# B&R Automation Studio project NAEUL004C00R13L518F00 (part 49)

#### Act_Main.st
```iecst
(** 2019-01-20 **)
ACTION Act_Main:

	IF eStatOld <> eStat THEN

		fbTxInTimer(IN := FALSE);
		fbTxOutTimer(IN := FALSE);
		fbMagOutTrig(CLK := FALSE);

		bMcRunRdy				 	  := FALSE;
		bRdyEnt			 		   	  := FALSE;
		bRdyExit				  	  := FALSE;
		bMagConvRun    := FALSE;
		fbCheckErrorTim(IN:= FALSE);
		usiStep		:= 0;

		sStatTxt	:= a_sStatText[eStat];

		eStatOld	:= eStat;

		eStatus		:= Busy;
	END_IF

	//Main
	CASE eStat OF

		AGVMagActIdle:
			eStatus	:= Idle;
			bMagConvRdy := FALSE;

		AGVMagActEnter:

			IF eStatus = Idle OR eStatus = Busy THEN

				eStatus	:= Busy;
				bMagConvRdy := TRUE;

				IF usiStep = 0 THEN

					IF bAIVAuto AND bMagConvAuto
						OR p_bSOTAvailable
						THEN // ON Connection

						bMagConvRdy  := TRUE; //Allow VEH to Move In

						IF bAIVInPos OR p_bSOTRcvOk THEN // VEH is in Position to Enter

							bRdyEnt := TRUE;

						END_IF
					END_IF

						IF bRdyEnt THEN

							IF bAIVInPos OR p_bSOTRcvOk  THEN

								bMagConvRdy := FALSE; // Temporarily Not Allowed Other VEH while one VEH in Pos.

								IF p_bSOTErr THEN
									eStatus		:= Error;
									udiStatus	:= 10010;//SOT Sensor Error Has Been Activated;

								ELSIF (NOT bMagConvOccupied) (*AND p_tyAGVToDTMag.bVEHOccupied*) THEN

									bMcRunRdy	:= TRUE;

									bMagConvRun := TRUE;

									usiStep	:= 1;
								ELSE
									eStatus		:= Error;
									udiStatus	:= 10000;	//Magazine Is Present Before Entering
								END_IF

							ELSE
								eStatus		:= Error;
								udiStatus	:= 10001;	//AIV Not In Enter Position
							END_IF

						END_IF

				ELSIF usiStep = 1 THEN

					IF p_eDirection = ConvDirLToL OR p_eDirection = ConvDirLToR THEN
						bEndSen	:= p_bMagConvRgtSen;
					ELSE
						bEndSen	:= p_bMagConvLftSen;
					END_IF

					fbTxInTimer(IN := TRUE, PT := DINT_TO_TIME(p_diTxInTimeOut));

					IF bEndSen = TRUE (*AND p_tyAGVToDTMag.bVEHOccupied = FALSE*) THEN

						eStatus	:= Done;

						bMagConvRdy := TRUE; // Allow VEH to Move Out After Transfering Magazine

						bMagConvRun := FALSE;

					ELSIF fbTxInTimer.Q = TRUE THEN

						eStatus		:= Error;
						udiStatus	:= 10002;	//Transfer In Time Out While Transporting

					END_IF

					IF bAIVInPos = FALSE AND p_bSOTRcvOk = FALSE AND eStatus = Busy THEN

						eStatus		:= Error;
						udiStatus	:= 10001;	//AIV Not In Enter Position
					END_IF

//					IF bAIVAuto = FALSE AND eStatus = Busy THEN
//
//						eStatus		:= Error;
//						udiStatus	:= 10006;	//AIV Not In Enter Position
//					END_IF
				END_IF

			END_IF

		AGVMagActExit:
			IF eStatus = Idle OR eStatus = Busy THEN

				eStatus	:= Busy;

				bMagConvRdy := TRUE;

				IF usiStep = 0 THEN

					IF bAIVAuto AND bMagConvAuto
						OR p_bSOTRdy
						THEN // ON Connection

						bMagConvRdy  := TRUE; //Allow VEH to Move In

						IF bAIVInPos OR p_bSOTRcvOk THEN // VEH is in Position to Exit

							bRdyExit := TRUE;

						END_IF
					END_IF

						IF bRdyExit THEN

							IF (bAIVInPos OR p_bSOTRcvOk) AND bAIVOccupied=FALSE THEN

								bMagConvRdy := FALSE; // Temporarily Not Allowed Other VEH while one VEH in Pos.

								IF bMagConvOccupied OR p_bSOTRdy = FALSE THEN

									bMcRunRdy	:= TRUE;

									bMagConvRun := TRUE;

									usiStep	:= 1;

								ELSE
									eStatus		:= Error;
									udiStatus	:= 10003;	//Magazine Is Not Present Before Exiting
								END_IF

							ELSE
								eStatus		:= Error;
								udiStatus	:= 10004;	//AIV Not In Exit Position
							END_IF
						END_IF

				ELSIF usiStep = 1 THEN

					IF p_bSOTErr THEN

						usiStep := 2;
					END_IF

					IF p_eDirection = ConvDirLToR OR p_eDirection = ConvDirRToR THEN
						bEndSen	:= p_bMagConvRgtSen;
					ELSE
						bEndSen	:= p_bMagConvLftSen;
					END_IF

					fbTxOutTimer(IN := TRUE, PT := DINT_TO_TIME(p_diTxOutTimeOut));

					IF bEndSen = FALSE AND (bAIVOccupied = TRUE OR p_bSOTRdy = FALSE) THEN

						usiStep := 2;

					ELSIF fbTxOutTimer.Q = TRUE THEN

						eStatus		:= Error;
						udiStatus	:= 10005;	//Transfer Out Time Out While Transporting

					END_IF

					IF bAIVInPos = FALSE AND p_bSOTRcvOk = FALSE AND eStatus = Busy THEN

						eStatus		:= Error;
						udiStatus	:= 10001;	//AIV Not In Enter Position
					END_IF

//					IF bAIVAuto = FALSE AND eStatus = Busy THEN
//
//						eStatus		:= Error;
//						udiStatus	:= 10006;	//AIV Not In Auto
//					END_IF

				ELSIF usiStep = 2 THEN
					fbCheckErrorTim(IN:= TRUE);
					IF p_bSOTErr THEN
						eStatus		:= Error;
						udiStatus	:= 10010;	//SOT Error signal activated
					ELSIF fbCheckErrorTim.Q THEN
						usiStep := 3;
					END_IF

				ELSIF usiStep = 3 THEN
					bMagConvRdy 	   := TRUE; // Allow VEH to Move Out After Transfering Magazine

					bMagConvRun := FALSE;
					eStatus := Done;
				END_IF

			END_IF
	END_CASE

END_ACTION
```

#### Act_OutputConfig.st
```iecst
ACTION Act_OutputConfig:

	g_tyAGV2 := tylocalAGV.Out; // Change the Global Naming According to the Physical Hardware Module

END_ACTION
```

#### Cyclic.st
```iecst
(** 2019-01-11 **)
PROGRAM _CYCLIC

	IF bInitialDone = FALSE THEN
		IF g_tyStartUp.bNtSettingsLoadDone = TRUE THEN
			bInitialDone	:= TRUE;
			Act_Initial;
		END_IF

	ELSE
		Act_InputConfig;
		IF (tylocalAGV.In.bPrep = TRUE) AND (tylocalAGV.In.bEn = TRUE) AND (tylocalAGV.In.bDis = FALSE) THEN
			Act_Link;
			Act_Background;
			Act_Main;
		ELSE
			IF tylocalAGV.Out.eStat <> AGVMagActIdle THEN
				eStatus	:= Done;
			ELSE
				eStatus	:= Idle;
			END_IF
		END_IF
		Act_OutputConfig;
		Act_Alarm;

	END_IF

END_PROGRAM
```

#### Init.st
```iecst
(** 2019-01-20 **)
PROGRAM _INIT

	(* Always Change If Project Change *)

	sProgNm	:= 'AGVMag 2';

	//Physical Configuration

	//Pass Address To Global Address For External Use
	//Action, State & Status
	p_AGVMag2Stat				:= ADR(eStat);
	p_AGVMag2Status				:= ADR(eStatus);
	p_AGVMag2StatTxt			:= ADR(sStatTxt);

	//Alarm
	p_AGVMag2AlmData			:= ADR(tyAlmData);

	//Output
	p_AGVMag2RdyEnter			:= ADR(bRdyEnt);
	p_AGVMag2RdyExit			:= ADR(bRdyExit);
	p_AGVMag2McRunRdy			:= ADR(bMcRunRdy);
	p_AGVMag2DTMagToAGV			:= ADR(tyDTMagToAGV);

	(* Always Change If Project Change *)

END_PROGRAM
```

### Program Logical/AGVCom/AGV3 (IEC, version 1.00.0) - 1.00.0 - NtSMEMA v5.00.0

#### Act_InputConfig.st - Change By Project
```iecst
ACTION Act_InputConfig:

	(* Always Change If Project Change *)

	//Pass Data To Link
	tylocalAGV.In.bLinkOpsRun := g_tyOps.bRun;

	tylocalAGV.In.tyLinkBufferStat := g_tyBuffer3.tyBufferStat;
	tylocalAGV.In.bLinkAGVOnline := g_tyAGV.bInternalAGVOnline;
	tylocalAGV.In.tyLinkAGVtoDTMag := g_tyAGV.tyAGVToDTMag;

	//Pass Data To Internal Use
//	tylocalAGV.In.eAct := g_tyOpsMagConvUL3AGVMagAct;
	tylocalAGV.In.udiRstErr	:= g_tyRstErrOut.udiRstErr;
	tylocalAGV.In.bPrep := g_tyNtParamCurr.bProjAGVPrep;
	tylocalAGV.In.sProgNm := g_tyNtParamCurr.sAGVMag3ProgNm;

	tylocalAGV.In.diTxInTimeOut := g_tyMcParam.tMag3ConvRunTmOut;
	tylocalAGV.In.diTxOutTimeOut := g_tyMcParam.tMag3ConvRunTmOut;

	tylocalAGV.In.eDirection := g_tyNtParamCurr.bProjMagConvDir;
	tylocalAGV.In.bBufferMagPresent := g_tyDInput.bMagPresentSen3;
	tylocalAGV.In.bMagConvLftSen := g_tyDInput.bMagPresentSen3;
	tylocalAGV.In.bMagConvRgtSen := g_tyDInput.bMagConvEntSen3;
	tylocalAGV.In.bMagConvMtrIn := g_tyMagConv2Clp3.bMtrSigOnOrLToR;
	tylocalAGV.In.bMagConvMtrOut := g_tyMagConv2Clp3.bMtrDirOrRToL;

	tylocalAGV.In.bAGVInPosSen1	:= g_tyDInput.bMag3AIVInPosSen1;
	tylocalAGV.In.bAGVInPosSen2	:= g_tyDInput.bMag3AIVInPosSen2;

	tylocalAGV.In.bNtParamAGVInPosSenPrep := g_tyNtParamCurr.bProjAIVInPosSenPrep;

	tylocalAGV.In.bSOTRcvOk := g_tyDInput.bSOT1Receive;
	tylocalAGV.In.bSOTErr := g_tyDInput.bSOT1AIVError;
	tylocalAGV.In.bSOTRdy := g_tyDInput.bSOT1AIVReady;
	tylocalAGV.In.bSOTAvailable := g_tyDInput.bSOT1AIVAvailable;
	tylocalAGV.In.bEn := g_tyMcParam.AGVComEn;

	IF g_tyNtParamCurr.bProjMag3ConvPrep THEN
		tylocalAGV.In.eAct := tyOpsMagConvUL1.eAGVMagAct;
	ELSE
		tylocalAGV.In.eAct := eAct;
	END_IF

	IF EDGENEG(g_tyOps.bRun) THEN
		tylocalAGV.In.eAct	:= AGVMagActIdle;
	END_IF
END_ACTION
```

#### Act_OutputConfig.st - Change By Project
```iecst
ACTION Act_OutputConfig:

	g_tyAGV3 := tylocalAGV.Out; // Change the Global Naming According to the Physical Hardware Module

END_ACTION
```

#### Act_Initial.st - Do Not Change!!!
```iecst
(** 2019-01-12 **)
ACTION Act_Initial:

	//Initial
	sStatTxt	:= a_sStatText[eStat];

	fbTxInTimer(IN := FALSE);
	fbTxOutTimer(IN := FALSE);
	fbMagOutTrig(CLK := FALSE);

	bMcRunRdy			:= FALSE;
	bRdyEnt			 	:= FALSE;
	bRdyExit			:= FALSE;
	bMagConvRun	    	:= FALSE;

END_ACTION
```

#### Act_Link.st - Change By Project
```iecst
(** 2018-12-08 **)
ACTION Act_Link:

	//Machine --> AGV ---> Communication On & Machine itself RUN Mode
	IF p_bLinkOpsRun = TRUE THEN

		tyDTMagToAGV.bCI3Auto := TRUE;
	ELSE
		tyDTMagToAGV.bCI3Auto	:= FALSE;
	END_IF

	tyDTMagToAGV.bCI3Occupied 			:= p_bBufferMagPresent OR p_bMagConvLftSen OR p_bMagConvRgtSen; // Magazine is present

	fbMagFullTm(IN:= p_bMagConvRgtSen = FALSE AND p_bBufferMagPresent = FALSE);
	IF p_bBufferMagPresent AND p_tyLinkBufferStat.bBffrFull THEN
		tyDTMagToAGV.bCI3MagazineFull		:=  TRUE;
	ELSIF fbMagFullTm.Q THEN
		tyDTMagToAGV.bCI3MagazineFull		:=  FALSE;
	END_IF

	IF p_bLinkAGVOnline THEN

		p_tyAGVToDTMag.bVEHAuto		:= p_tyLinkAGVtoDTMag.bVEHAuto;
		p_tyAGVToDTMag.bVEHInPos1	:= p_tyLinkAGVtoDTMag.bVEHInPos1 AND bAGVInPosSen;
		p_tyAGVToDTMag.bVEHInPos2 	:= p_tyLinkAGVtoDTMag.bVEHInPos2;
		p_tyAGVToDTMag.bVEHInPos3 	:= p_tyLinkAGVtoDTMag.bVEHInPos3;
		p_tyAGVToDTMag.bVEH1Occupied	:= p_tyLinkAGVtoDTMag.bVEH1Occupied;
		p_tyAGVToDTMag.bVEH2Occupied	:= p_tyLinkAGVtoDTMag.bVEH2Occupied;
		p_tyAGVToDTMag.bVEH3Occupied	:= p_tyLinkAGVtoDTMag.bVEH3Occupied;
		p_tyAGVToDTMag.bVEHRunning	:= p_tyLinkAGVtoDTMag.bVEHRunning;

	ELSE

		p_tyAGVToDTMag.bVEHAuto		:= FALSE;
		p_tyAGVToDTMag.bVEHInPos1	:= FALSE;
		p_tyAGVToDTMag.bVEHInPos2 	:= FALSE;
		p_tyAGVToDTMag.bVEHInPos3 	:= FALSE;
		p_tyAGVToDTMag.bVEH1Occupied:= FALSE;
		p_tyAGVToDTMag.bVEH2Occupied:= FALSE;
		p_tyAGVToDTMag.bVEH3Occupied:= FALSE;
		p_tyAGVToDTMag.bVEHRunning	:= FALSE;

	END_IF

	bAIVInPos := p_tyAGVToDTMag.bVEHInPos3;
	bAIVAuto := p_tyAGVToDTMag.bVEHAuto;
	bAIVOccupied := p_tyAGVToDTMag.bVEH3Occupied;
	bMagConvAuto := tyDTMagToAGV.bCI3Auto;
	bMagConvOccupied :=  tyDTMagToAGV.bCI3Occupied;

	tyDTMagToAGV.bCI3Running := bMagConvRun;
	tyDTMagToAGV.bCI3Rdy	:= bMagConvRdy;

	IF p_bNtParamAGVInPosSenPrep THEN
		fbInPosErrTimer(IN:= p_tyLinkAGVtoDTMag.bVEHInPos3 AND bAGVInPosSen = FALSE, PT:= T#10s);
		IF fbInPosErrTimer.Q THEN
			eStatus		:= Error;
			udiStatus	:= 10009;	//AIV Not In Position
		END_IF
	END_IF

	IF p_bNtParamAGVInPosSenPrep THEN
		bAGVInPosSen := p_bAGVInPosSen1 AND p_bAGVInPosSen2;
	ELSE
		bAGVInPosSen := TRUE;
	END_IF

END_ACTION
```

#### Act_Main.st - Do Not Change!!!
```iecst
(** 2019-01-20 **)
ACTION Act_Main:

	//Set tylocalAGV.In.eAct
	IF tylocalAGV.Out.eStatus = Idle OR tylocalAGV.Out.eStatus = Busy OR tylocalAGV.Out.eStatus = Done THEN
		tylocalAGV.Out.eStat	:= tylocalAGV.In.eAct;
	END_IF

	IF eStatOld <> tylocalAGV.Out.eStat THEN

		fbTxInTimer(IN := FALSE);
		fbTxOutTimer(IN := FALSE);
		fbMagOutTrig(CLK := FALSE);

		tylocalAGV.Out.bMcRunRdy				 	  := FALSE;
		tylocalAGV.Out.bRdyEnt			 		   	  := FALSE;
		tylocalAGV.Out.bRdyExit				  	  := FALSE;
		bMagConvRun    := FALSE;
		fbCheckErrorTim(IN:= FALSE);
		usiStep		:= 0;

		tylocalAGV.Out.sStatTxt	:= a_sStatText[tylocalAGV.Out.eStat];

		eStatOld	:= tylocalAGV.Out.eStat;

		tylocalAGV.Out.eStatus		:= Busy;
	END_IF

	//Main
	CASE tylocalAGV.Out.eStat OF

		AGVMagActIdle:
			tylocalAGV.Out.eStatus	:= Idle;
			bMagConvRdy := FALSE;

		AGVMagActEnter:

			IF tylocalAGV.Out.eStatus = Idle OR tylocalAGV.Out.eStatus = Busy THEN

				tylocalAGV.Out.eStatus	:= Busy;
				bMagConvRdy := TRUE;

				IF usiStep = 0 THEN

					IF bAIVAuto AND bMagConvAuto
						OR tylocalAGV.In.bSOTAvailable
						THEN // ON Connection

						bMagConvRdy  := TRUE; //Allow VEH to Move In

						IF bAIVInPos OR tylocalAGV.In.bSOTRcvOk THEN // VEH is in Position to Enter

							tylocalAGV.Out.bRdyEnt := TRUE;

						END_IF
					END_IF

						IF tylocalAGV.Out.bRdyEnt THEN

							IF bAIVInPos OR tylocalAGV.In.bSOTRcvOk  THEN

								bMagConvRdy := FALSE; // Temporarily Not Allowed Other VEH while one VEH in Pos.

								IF tylocalAGV.In.bSOTErr THEN
									tylocalAGV.Out.eStatus		:= Error;
									udiStatus	:= 10010;//SOT Sensor Error Has Been Activated;

								ELSIF (NOT bMagConvOccupied) (*AND tylocalAGV.In.tyAGVToDTMag.bVEHOccupied*) THEN

									tylocalAGV.Out.bMcRunRdy	:= TRUE;

									bMagConvRun := TRUE;

									usiStep	:= 1;
								ELSE
									tylocalAGV.Out.eStatus		:= Error;
									udiStatus	:= 10000;	//Magazine Is Present Before Entering
								END_IF

							ELSE
								tylocalAGV.Out.eStatus		:= Error;
								udiStatus	:= 10001;	//AIV Not In Enter Position
							END_IF

						END_IF

				ELSIF usiStep = 1 THEN

					IF tylocalAGV.In.eDirection = ConvDirLToL OR tylocalAGV.In.eDirection = ConvDirLToR THEN
						bEndSen	:= tylocalAGV.In.bMagConvRgtSen;
					ELSE
						bEndSen	:= tylocalAGV.In.bMagConvLftSen;
					END_IF

					fbTxInTimer(IN := TRUE, PT := DINT_TO_TIME(tylocalAGV.In.diTxInTimeOut));

					IF bEndSen = TRUE (*AND tylocalAGV.In.tyAGVToDTMag.bVEHOccupied = FALSE*) THEN

						tylocalAGV.Out.eStatus	:= Done;

						bMagConvRdy := TRUE; // Allow VEH to Move Out After Transfering Magazine

						bMagConvRun := FALSE;

					ELSIF fbTxInTimer.Q = TRUE THEN

						tylocalAGV.Out.eStatus		:= Error;
						udiStatus	:= 10002;	//Transfer In Time Out While Transporting

					END_IF

					IF bAIVInPos = FALSE AND tylocalAGV.In.bSOTRcvOk = FALSE AND tylocalAGV.Out.eStatus = Busy THEN

						tylocalAGV.Out.eStatus		:= Error;
						udiStatus	:= 10001;	//AIV Not In Enter Position
					END_IF

//					IF bAIVAuto = FALSE AND tylocalAGV.Out.eStatus = Busy THEN
//
//						tylocalAGV.Out.eStatus		:= Error;
//						udiStatus	:= 10006;	//AIV Not In Enter Position
//					END_IF
				END_IF

			END_IF

		AGVMagActExit:
			IF tylocalAGV.Out.eStatus = Idle OR tylocalAGV.Out.eStatus = Busy THEN

				tylocalAGV.Out.eStatus	:= Busy;

				bMagConvRdy := TRUE;

				IF usiStep = 0 THEN

					IF bAIVAuto AND bMagConvAuto
						OR tylocalAGV.In.bSOTRdy
						THEN // ON Connection

						bMagConvRdy  := TRUE; //Allow VEH to Move In

						IF bAIVInPos OR tylocalAGV.In.bSOTRcvOk THEN // VEH is in Position to Exit

							tylocalAGV.Out.bRdyExit := TRUE;

						END_IF
					END_IF

						IF tylocalAGV.Out.bRdyExit THEN

							IF (bAIVInPos OR tylocalAGV.In.bSOTRcvOk) AND bAIVOccupied=FALSE THEN

								bMagConvRdy := FALSE; // Temporarily Not Allowed Other VEH while one VEH in Pos.

								IF bMagConvOccupied OR tylocalAGV.In.bSOTRdy = FALSE THEN

									tylocalAGV.Out.bMcRunRdy	:= TRUE;

									bMagConvRun := TRUE;

									usiStep	:= 1;

								ELSE
									tylocalAGV.Out.eStatus		:= Error;
									udiStatus	:= 10003;	//Magazine Is Not Present Before Exiting
								END_IF

							ELSE
								tylocalAGV.Out.eStatus		:= Error;
								udiStatus	:= 10004;	//AIV Not In Exit Position
							END_IF
						END_IF

				ELSIF usiStep = 1 THEN

					IF tylocalAGV.In.bSOTErr THEN

						usiStep := 2;
					END_IF

					IF tylocalAGV.In.eDirection = ConvDirLToR OR tylocalAGV.In.eDirection = ConvDirRToR THEN
						bEndSen	:= tylocalAGV.In.bMagConvRgtSen;
					ELSE
						bEndSen	:= tylocalAGV.In.bMagConvLftSen;
					END_IF

					fbTxOutTimer(IN := TRUE, PT := DINT_TO_TIME(tylocalAGV.In.diTxOutTimeOut));

					IF bEndSen = FALSE AND (bAIVOccupied = TRUE OR tylocalAGV.In.bSOTRdy = FALSE) THEN

						usiStep := 2;

					ELSIF fbTxOutTimer.Q = TRUE THEN

						tylocalAGV.Out.eStatus		:= Error;
						udiStatus	:= 10005;	//Transfer Out Time Out While Transporting

					END_IF

					IF bAIVInPos = FALSE AND tylocalAGV.In.bSOTRcvOk = FALSE AND tylocalAGV.Out.eStatus = Busy THEN

						tylocalAGV.Out.eStatus		:= Error;
						udiStatus	:= 10001;	//AIV Not In Enter Position
					END_IF

//					IF bAIVAuto = FALSE AND tylocalAGV.Out.eStatus = Busy THEN
//
//						tylocalAGV.Out.eStatus		:= Error;
//						udiStatus	:= 10006;	//AIV Not In Auto
//					END_IF

				ELSIF usiStep = 2 THEN
					fbCheckErrorTim(IN:= TRUE);
					IF tylocalAGV.In.bSOTErr THEN
						tylocalAGV.Out.eStatus		:= Error;
						udiStatus	:= 10010;	//SOT Error signal activated
					ELSIF fbCheckErrorTim.Q THEN
						usiStep := 3;
					END_IF

				ELSIF usiStep = 3 THEN
					bMagConvRdy 	   := TRUE; // Allow VEH to Move Out After Transfering Magazine

					bMagConvRun := FALSE;
					tylocalAGV.Out.eStatus := Done;
				END_IF

			END_IF
	END_CASE

END_ACTION
```

#### Act_Alarm.st - Do Not Change!!!
```iecst
(** 2019-03-25 **)
ACTION Act_Alarm:

	//Error
	IF EDGEPOS(eStatus = Error) THEN

		tyAlmData.sProgNm		:= p_sProgNm;
		tyAlmData.udiCode		:= udiStatus;
		tyAlmData.eSeverity		:= AlmSeverityError;
		tyAlmData.udiRunTime	:= tyAlmData.udiRunTime + 1;
		tyAlmData.bAlm			:= TRUE;
		tyAlmData.udiModuleNum  := udiModuleNum;
		g_sAGVProgNm		:= p_sProgNm;

		//Get Error Message
		IF tyAlmData.udiCode < 10000 OR tyAlmData.udiCode > 10099 THEN
			tyAlmData.sAlmMsg	:= 'Unknown';
			tyAlmData.sRcyMsg	:= 'Unknown';
		ELSE
			tyAlmData.sAlmMsg	:= a_tyAlmText[tyAlmData.udiCode].sAlmText;
			tyAlmData.sRcyMsg	:= a_tyAlmText[tyAlmData.udiCode].sRcyText;
		END_IF

		sStatTxt	:= tyAlmData.sAlmMsg;

	ELSIF bRstErr AND (tyAlmData.udiCode <> 0) THEN

		tyAlmData.udiCode	:= 0;
		tyAlmData.eSeverity	:= AlmSeverityNA;
		tyAlmData.sAlmMsg	:= '';
		tyAlmData.sRcyMsg	:= '';

		sStatTxt	:= a_sStatText[eStat];

	END_IF

END_ACTION
```

#### Cyclic.st - Do Not Change!!!
```iecst
(** 2019-01-11 **)
PROGRAM _CYCLIC

	IF bInitDone = FALSE THEN
		bInitDone	:= TRUE;

		Act_InitLocal;
		Act_InitGlobal;

	ELSIF bInitialDone = FALSE THEN
		IF p_bNtSettingsLoadDone = TRUE THEN
			bInitialDone	:= TRUE;

			Act_Initial;
		END_IF

	ELSE

		Act_RstErr;
		Act_LinkAction;
		Act_Action;
		Act_LinkEn;

		IF (p_bPrep = TRUE) AND (p_bEn = TRUE) AND (p_bDis = FALSE) THEN
			Act_Link;
			Act_Background;
			Act_Main;
		ELSE
			IF eStat <> AGVMagActIdle THEN
				eStatus	:= Done;
			ELSE
				eStatus	:= Idle;
			END_IF
		END_IF

		Act_Alarm;

	END_IF

END_PROGRAM
```

#### Local.var - Do Not Change!!!
```iecst
(*2019-01-20*)
(**)
(*Local Action, State & Status*)
VAR
	eAct : eAGVMagAction := AGVMagActIdle;
	eStat : eAGVMagAction := AGVMagActIdle;
	eStatus : eFBStatus := Idle;
	udiStatus : UDINT := 0;
	sStatTxt : STRING[100] := '';
	a_sStatText : ARRAY[0..50] OF STRING[100] := ['Idling','AIV Magazine Ready Enter And Communicating AIV','AIV Magazine Ready Exit And Communicating AIV',48('')];
END_VAR
(**)
(*Local Alarm*)
VAR
	tyAlmData : tyAlmDat;
	a_tyAlmText : ARRAY[10000..10099] OF tyAlmTxt := [(sAlmText:='Magazine Is Present Before Entering',sRcyText:='Remove Magazine To Continue Operation.'),(sAlmText:='AGV Not In Enter Position',sRcyText:='Adjust AGV Position And Restart Operation.'),(sAlmText:='Transfer In Time Out While Transporting',sRcyText:='Adjust Magazine Position Or Transporting Time Or Check Online Connection'),(sAlmText:='Magazine Is Not Present Before Exiting',sRcyText:='Magazine Has Taken Away, Restart Operation.'),(sAlmText:='AGV Not In Exit Position',sRcyText:='Adjust AGV Position And Restart Operation.'),(sAlmText:='Transfer Out Time Out While Transporting',sRcyText:='Adjust Magazine Position Or Transporting Time.'),(sAlmText:='AGV is not in Auto',sRcyText:='Make Sure AGV is in Auto'),(sAlmText:='Magazine is not Present in AGV while Entering',sRcyText:='Check AGV'),(sAlmText:='Magazine is Present in AGV while Exiting',sRcyText:='Check AGV'),(sAlmText:='AGV In Position Sensor is off while received the AGV in position signal',sRcyText:='Check AGV in position sensor'),(sAlmText:='SOT Error Signal Has Been Activated',sRcyText:='AIV Activated The Error Signal During Magazine Transportation'),89((0))];
END_VAR
(**)
(*Local Output*)
VAR
	bMcRunRdy : BOOL;
	bRdyEnt : BOOL;
	bRdyExit : BOOL;
	bMagEnt : BOOL;
	bMagExit : BOOL;
END_VAR
(**)
(*Local Input*)
VAR
	udiRstErr : UDINT := 0;
	bPrep : BOOL := TRUE;
	bEn : BOOL := TRUE;
	bDis : BOOL := FALSE;
	sProgNm : STRING[15] := 'AIVMag';
	bNtSettingsLoadDone : BOOL := TRUE;
	diTxInTimeOut : DINT;
	diTxOutTimeOut : DINT;
	eDirection : eConvDir;
	bBufferMagPresent : BOOL;
	bMagConvLftSen : BOOL;
	bMagConvRgtSen : BOOL;
	bMagConvMtrIn : BOOL;
	bMagConvMtrOut : BOOL;
	bAGVInPosSen1 : BOOL;
	bAGVInPosSen2 : BOOL;
	bNtParamAGVInPosSenPrep : BOOL;
	tyAGVToDTMag : tyTagAGVToDTMag;
	tyDTMagToAGV : tyTagDTMagToAGV;
END_VAR
(**)
(*Local*)
VAR
	bRstErr : BOOL;
	udiRstErrOld : UDINT;
	bInitDone : BOOL;
	bInitialDone : BOOL;
	usiStep : USINT;
	bEndSen : BOOL;
	bAGVInPosSen : BOOL;
	fbMagFullTm : TON := (PT:=T#2s);
	fbInPosErrTimer : TON;
	fbTxInTimer : TON;
	fbTxOutTimer : TON;
	fbMagOutTrig : F_TRIG;
	eStatOld : eAGVMagAction := AGVMagActIdle;
	fbCheckErrorTim : TON := (PT:=T#1s);
	bMagConvRun : BOOL;
	bMagConvRdy : BOOL;
	bMagConvAuto : BOOL;
	bMagConvOccupied : BOOL;
	bAIVOccupied : BOOL;
	bAIVAuto : BOOL;
	bAIVInPos : BOOL;
	udiModuleNum : UDINT := 6161;
END_VAR
```

#### InputRef_Link.var - not listed in the package file held
```iecst
(*2018-12-08*)
(**)
(*External Data*)
VAR
	p_bLinkAGVOnline : REFERENCE TO BOOL;
	p_bLinkOpsRun : REFERENCE TO BOOL;
END_VAR
(**)
VAR
	p_tyLinkBufferStat : REFERENCE TO tyBffrStat;
	p_tyLinkAGVtoDTMag : REFERENCE TO tyTagAGVToDTMag;
	p_bLinkProjMag3ConvPrep : REFERENCE TO BOOL;
END_VAR
```

#### Act_InitGlobal.st - not listed in the package file held
```iecst
(** 2018-12-08 **)
ACTION Act_InitGlobal:

	(* Always Change If Project Change *)

	//Pass Data To Link
	p_bLinkOpsRun ACCESS p_OpsRun;

	p_tyLinkBufferStat ACCESS p_Buffer3BffrStat;
	p_bLinkAGVOnline ACCESS p_AGVOnline;
	p_tyLinkAGVtoDTMag ACCESS p_AGVTagAGVToDTMag;
	p_bLinkProjMag3ConvPrep ACCESS p_NtParamProjMag3ConvPrep;

	//Pass Data To Internal Use
	p_eAct ACCESS p_OpsMagConvUL3AGVMagAct;
	p_udiRstErr	ACCESS p_RstErrReset;
	p_bPrep ACCESS p_NtParamProjAGVPrep;
	p_sProgNm ACCESS p_NtParamAGVMag3ProgNm;
	p_diTxInTimeOut ACCESS p_McParamMag3ConvRunTmOut;
	p_diTxOutTimeOut ACCESS p_McParamMag3ConvRunTmOut;
	p_eDirection ACCESS p_NtParamProjMagConvDir;
	p_bBufferMagPresent ACCESS p_DIMagPresentSen3;
	p_bMagConvLftSen ACCESS p_DIMagPresentSen3;
	p_bMagConvRgtSen ACCESS p_DIMagConvEntSen3;
	p_bMagConvMtrIn ACCESS p_MagConv2Clp1MtrSigOnOrLToR;
	p_bMagConvMtrOut ACCESS p_MagConv2Clp1MtrDirOrRToL;
	p_bNtSettingsLoadDone ACCESS p_StartupNtSettingsLoadDone;
	p_bAGVInPosSen1	ACCESS p_DIMag3AIVInPosSen1;
	p_bAGVInPosSen2	ACCESS p_DIMag3AIVInPosSen2;
	p_bNtParamAGVInPosSenPrep ACCESS p_NtParamProjAIVInPosSenPrep;
	p_bSOTRcvOk ACCESS p_DISOT3Receive;
	p_bSOTErr ACCESS p_DISOT3Error;
	p_bSOTRdy ACCESS p_DISOT3Ready;
	p_bSOTAvailable ACCESS p_DISOT3Available;
	p_bEn ACCESS p_McParamAGVComEn;
	(* Always Change If Project Change *)

END_ACTION
```

#### Act_LinkAction.st - not listed in the package file held
```iecst
(** 2019-03-29 **)
ACTION Act_LinkAction:

	IF EDGENEG(p_bLinkOpsRun) THEN
		p_eAct	:= AGVMagActIdle;
	END_IF

END_ACTION
```

#### Init.st - not listed in the package file held
```iecst
(** 2019-01-20 **)
PROGRAM _INIT

	(* Always Change If Project Change *)

	sProgNm	:= 'AGVMag 3';

	//Physical Configuration

	//Pass Address To Global Address For External Use
	//Action, State & Status
	p_AGVMag3Stat		:= ADR(eStat);
	p_AGVMag3Status		:= ADR(eStatus);
	p_AGVMag3StatTxt	:= ADR(sStatTxt);

	//Alarm
	p_AGVMag3AlmData	:= ADR(tyAlmData);

	//Output
	p_AGVMag3RdyEnter		:= ADR(bRdyEnt);
	p_AGVMag3RdyExit		:= ADR(bRdyExit);
	p_AGVMag3McRunRdy		:= ADR(bMcRunRdy);
	p_AGVMag3DTMagToAGV		:= ADR(tyDTMagToAGV);

	(* Always Change If Project Change *)

END_PROGRAM
```

### AGV1.var - not listed in the package file held
```iecst
(*2019-01-20*)
(**)
(*Action & State & Status*)
VAR
	p_AGVMag1Stat : UDINT;
	p_AGVMag1Status : UDINT;
	p_AGVMag1StatTxt : UDINT;
END_VAR
(**)
(*Alarm*)
VAR
	p_AGVMag1AlmData : UDINT;
END_VAR
(**)
(*Output*)
VAR
	p_AGVMag1RdyEnter : UDINT;
	p_AGVMag1RdyExit : UDINT;
	p_AGVMag1McRunRdy : UDINT;
	p_AGVMag1Exit : UDINT;
	p_AGVMag1DTMagToAGV : UDINT;
END_VAR
```

### AGV2.var - not listed in the package file held
```iecst
(*2019-01-20*)
(**)
(*Action & State & Status*)
VAR
	p_AGVMag2Stat : UDINT;
	p_AGVMag2Status : UDINT;
	p_AGVMag2StatTxt : UDINT;
END_VAR
(**)
(*Alarm*)
VAR
	p_AGVMag2AlmData : UDINT;
END_VAR
(**)
(*Output*)
VAR
	p_AGVMag2RdyEnter : UDINT;
	p_AGVMag2RdyExit : UDINT;
	p_AGVMag2McRunRdy : UDINT;
	p_AGVMag2Exit : UDINT;
	p_AGVMag2DTMagToAGV : UDINT;
END_VAR
```

### AGV3.var - not listed in the package file held
```iecst
(*2019-01-20*)
(**)
(*Action & State & Status*)
VAR
	p_AGVMag3Stat : UDINT;
	p_AGVMag3Status : UDINT;
	p_AGVMag3StatTxt : UDINT;
END_VAR
(**)
(*Alarm*)
VAR
	p_AGVMag3AlmData : UDINT;
END_VAR
(**)
(*Output*)
VAR
	p_AGVMag3RdyEnter : UDINT;
	p_AGVMag3RdyExit : UDINT;
	p_AGVMag3McRunRdy : UDINT;
	p_AGVMag3Exit : UDINT;
	p_AGVMag3DTMagToAGV : UDINT;
END_VAR
```

### AW.typ - Do Not Change!!!
```iecst
(*2019-01-24*)
(**)
(*Action*)

TYPE
	eAWAction :
		(
		AWActIdle,
		AWActGoWidth,
		AWActFullHm,
		AWActPwrOn,
		AWActPwrOff,
		AWActHoming,
		AWActMovAbs,
		AWActMovRel,
		AWActJogOpen,
		AWActJogClose,
		AWActJogStop,
		AWActRstAxisErr,
		AWActStop,
		AWActSDOWrite,
		AWActBGStartModOKChk,
		AWActBGStopModOKChk,
		AWActGoWidthOff,
		AWActRstNode
		);
END_TYPE
```

### Program Logical/CANOpenServo/AW/AWOpen (IEC, version 1.00.0) - 1.00.0 - NtMotion v5.00.0

#### Init.st - Change By Project
```iecst
(** 2019-04-24 **)
PROGRAM _INIT

	(* Always Change If Project Change *)

	//Pass Address To Global Address For External Use
	//Action, State & Status
	p_AWOpenStat	:= ADR(eStat);
	p_AWOpenStatus	:= ADR(eMainStatus);
	p_AWOpenStatTxt	:= ADR(sStatTxt);

	//Alarm
	p_AWOpenAlmData		:= ADR(tyAlmData);
	p_AWOpenAlmData1	:= ADR(tyAlmData1);
	p_AWOpenAlmData2	:= ADR(tyAlmData2);
	p_AWOpenAlmData3	:= ADR(tyAlmData3);

	//Output
	p_AWOpenParamOut		:= ADR(tyParamOut);
	p_AWOpenPwrOn			:= ADR(tyParamOut.bPwrOn);
	p_AWOpenIsHomed			:= ADR(tyParamOut.bIsHomed);
	p_AWOpenPosDiff			:= ADR(tyParamOut.bPosDiff);
	p_AWOpenAxisErr			:= ADR(tyParamOut.bAxisErr);
	p_AWOpenAxisErrID		:= ADR(tyParamOut.udiAxisErrID);
	p_AWOpenFwdLmtSen		:= ADR(tyParamOut.bFwdLmtSen);
	p_AWOpenRevLmtSen		:= ADR(tyParamOut.bRevLmtSen);
	p_AWOpenActualPos		:= ADR(tyParamOut.diActualPosInUM);
	p_AWOpenAxisErrTxt		:= ADR(sAxisErrTxt);
	p_AWOpenWidthPosDiff	:= ADR(bWidthPosDiff);
	p_AWOpenJogging			:= ADR(bJogging);
	p_AWOpenOpenSen			:= ADR(bOpenSen);
	p_AWOpenCloseSen		:= ADR(bCloseSen);

	(* Always Change If Project Change *)

END_PROGRAM
```

#### Act_InitGlobal.st - Change By Project
```iecst
(** 2019-04-09 **)
ACTION Act_InitGlobal:

	(* Always Change If Project Change *)

	//Pass Data To Link
	p_bLinkOpsRun ACCESS p_OpsRun;
	p_bLinkStartupRun ACCESS p_StartupRun;
	p_bLinkSafetyRelay ACCESS p_DISafetyRlySig;
	//Pass Data To Internal Use
	p_udiRstErr ACCESS p_RstErrReset;
	p_bPrep ACCESS p_NtParamAWPrep;
	p_bDis ACCESS p_McParamAWDis;
	p_bOps ACCESS p_OpsStatusRun;
	p_bManual ACCESS p_UIMnlMod;
	p_diWidthAtHmPos ACCESS p_McParamWidthAtHmPos;
	p_tyTuning ACCESS p_NtParamAWTuning;
	p_diJogVelInUMPS ACCESS p_UIMnlAWJogSpd;
	p_diMovePosInUM ACCESS p_UIMnlAWTargetPos;
	p_diMoveDistInUM ACCESS p_UIMnlAWStepSize;
	p_diMoveAcc ACCESS p_NtParamAWAcc;
	p_diMoveDec ACCESS p_NtParamAWDec;
	p_diMinWidthInUM ACCESS p_NtParamProdRcpMinWidth;
	p_diMaxWidthInUM ACCESS p_NtParamProdRcpMaxWidth;
	p_diWidthOffsetInUM ACCESS p_NtParamWidthOffset;
	p_bInletSensor ACCESS p_DIConvLftSen;
	p_bOutletSensor ACCESS p_DIConvRgtSen;
	p_bClearSensor ACCESS p_DIConvClrSen;
	p_bMiddleSensor ACCESS p_DIConvMidSen;
	p_bDir ACCESS p_NtParamAWDir;
	p_bDirBl ACCESS p_NtParamAWDirBl;
	p_usiNode ACCESS p_NtParamAWNode;
	p_sDevice ACCESS p_NtParamAWDevice;
	p_sProgNm ACCESS p_NtParamAWProgNm;
	p_diMoveBacklashDistInUM ACCESS p_NtParamAWMovBlDistInUM;
	p_diPitchInUM ACCESS p_NtParamAWPitchInUM;
	p_tyParamInHm ACCESS p_NtParamAWParamInHm;
	p_tyParamInConvert ACCESS p_NtParamAWParamInConvert;
	p_bNtSettingsLoadDone ACCESS p_StartupNtSettingsLoadDone;
	p_eNtParamMotorType ACCESS p_NtParamAWMotorType;

	p_bInletShutterCloseRS ACCESS p_DIInShutterCloseRS;
	p_bOutletShutterCloseRS ACCESS p_DIOutShutterCloseRS;
	p_bOutletShutterCloseRS2 ACCESS p_DIOutShutterCloseRS2;
	p_bOutletShutterCloseRS3 ACCESS p_DIOutShutterCloseRS3;
	p_bProjInletShutPrep ACCESS p_NtParamProjInletShutPrep;
	p_bInShutterDis ACCESS p_McParamInShutterDis;
	p_bProjOutletShutPrep ACCESS p_NtParamProjOutletShutPrep;

	p_bPusherRetSen ACCESS p_DIPusherRetRS;
	p_bPusherExtSen ACCESS p_DIPusherExtRS;

	p_bNtParamAutoRcpPrep ACCESS p_NtParamAutoRcpPrep ;
	p_bMcParamAutoRcpDis  ACCESS p_McParamAutoRcpDisable;
	p_eNtParamAutoRcpPrecededBy ACCESS p_NtParamAutoRcpPrecededBy;
	//follower action link to rcp1 but can use with smeama
	(* Always Change If Project Change *)

END_ACTION
```

#### InputRef_Link.var - Change By Project
```iecst
(*2019-04-09*)
(**)
(*External Data*)
VAR
	p_bLinkOpsRun : REFERENCE TO BOOL;
	p_bLinkStartupRun : REFERENCE TO BOOL;
	p_bLinkSafetyRelay : REFERENCE TO BOOL;
END_VAR
```

#### Act_LinkAction.st - Change By Project
```iecst
(** 2019-10-21 **)
ACTION Act_LinkAction:

	IF eStatus = Idle THEN
		IF bModuleNotOK THEN
			p_eAct ACCESS ADR(eAct);
		ELSE
			IF p_bLinkStartupRun = TRUE THEN
				p_eAct ACCESS p_StartupAWAct;
			ELSIF p_bLinkOpsRun = TRUE THEN
				p_eAct ACCESS p_OpsTravLifULAWAct;
			ELSIF p_bManual = TRUE THEN
				p_eAct ACCESS p_UIAWOpenAct;
			ELSE
				p_eAct ACCESS ADR(eAct);
			END_IF
		END_IF
	END_IF

	IF EDGENEG(p_bManual) OR EDGENEG(p_bLinkOpsRun) OR EDGENEG(p_bLinkStartupRun) THEN
		tyParamOutDriver.uiCtrlword_6040	:= 0;
	END_IF

END_ACTION
```

#### Act_Link.st - Change By Project
```iecst
(** 2019-03-29 **)
ACTION Act_Link:

	IF p_bManual = TRUE THEN
		p_diGoWidth ACCESS p_UIMnlAWGoWidth;
		p_diMoveVelInUMPS ACCESS p_UIMnlAWNomSpd;
	ELSE
		IF p_bNtParamAutoRcpPrep AND NOT(p_bMcParamAutoRcpDis)  THEN
			CASE p_eNtParamAutoRcpPrecededBy OF
				PrecededBySelf:
					p_diGoWidth ACCESS p_diAutoRcpTravLifWidth;
				PrecededByF1:
					p_diGoWidth ACCESS p_ProdRcpCurrRcp1Width;
			END_CASE
		ELSE
			p_diGoWidth ACCESS p_ProdRcpCurrRcp1Width;
		END_IF
		p_diMoveVelInUMPS ACCESS p_NtParamAWAutoSpd;
	END_IF

	IF p_bProjInletShutPrep = TRUE AND p_bInShutterDis = FALSE AND (p_bOps OR p_bManual) THEN
		IF (p_bInletShutterCloseRS = FALSE AND NOT p_bOps) OR p_bPusherRetSen = FALSE OR p_bPusherExtSen THEN
			bInterruptSensor1 := TRUE;
		ELSE
			bInterruptSensor1 := FALSE;
		END_IF
	ELSE
		bInterruptSensor1 := FALSE;
	END_IF

	IF p_bProjOutletShutPrep = TRUE AND (p_bOps OR p_bManual)THEN
		IF ((p_bOutletShutterCloseRS = FALSE OR p_bOutletShutterCloseRS2 = FALSE OR p_bOutletShutterCloseRS3 = FALSE) AND NOT p_bOps) OR p_bPusherRetSen = FALSE OR p_bPusherExtSen THEN
			bInterruptSensor2 := TRUE;
		ELSE
			bInterruptSensor2 := FALSE;
		END_IF
	ELSE
		bInterruptSensor2 := FALSE;
	END_IF

	IF NOT p_bOps THEN
		bInterruptSensor1	:= FALSE;
		bInterruptSensor2   := FALSE;
		p_bInterruptSensor	:= FALSE;
	END_IF

	p_bInterruptSensor := bInterruptSensor2 OR bInterruptSensor1;// OR p_bLinkSafetyRelay = FALSE;

END_ACTION
```

#### Act_InitLocal.st - Change By Project
```iecst
(** 2020-05-26 **)
ACTION Act_InitLocal:

	//Input Reference Link To Local Variable
	p_eAct ACCESS ADR(eAct);
	p_udiRstErr ACCESS ADR(udiRstErr);
	p_bPrep ACCESS ADR(bPrep);
	p_bEn ACCESS ADR(bEn);
	p_bDis ACCESS ADR(bDis);
	p_bOps ACCESS ADR(bOps);
	p_bManual ACCESS ADR(bManual);
	p_diWidthAtHmPos ACCESS ADR(diWidthAtHmPos);
	p_tyTuning ACCESS ADR(tyTuning);
	p_diGoWidth ACCESS ADR(diGoWidth);
	p_diJogVelInUMPS ACCESS ADR(diJogVelInUMPS);
	p_diMovePosInUM ACCESS ADR(diMovePosInUM);
	p_diMoveDistInUM ACCESS ADR(diMoveDistInUM);
	p_diMoveVelInUMPS ACCESS ADR(diMoveVelInUMPS);
	p_diMoveAcc ACCESS ADR(diMoveAcc);
	p_diMoveDec ACCESS ADR(diMoveDec);
	p_diMinAbsPosInUM ACCESS ADR(diMinAbsPosInUM);
	p_diMaxAbsPosInUM ACCESS ADR(diMaxAbsPosInUM);
	p_diMinWidthInUM ACCESS ADR(diMinWidthInUM);
	p_diMaxWidthInUM ACCESS ADR(diMaxWidthInUM);
	p_diWidthOffsetInUM ACCESS ADR(diWidthOffsetInUM);
	p_bInletSensor ACCESS ADR(bInletSensor);
	p_bOutletSensor ACCESS ADR(bOutletSensor);
	p_bClearSensor ACCESS ADR(bClearSensor);
	p_bMiddleSensor ACCESS ADR(bMiddleSensor);
	p_bInterruptSensor ACCESS ADR(bInterruptSensor);
	p_bOpenInterruptSensor ACCESS ADR(bOpenInterruptSensor);
	p_bCloseInterruptSensor ACCESS ADR(bCloseInterruptSensor);
	p_bDir ACCESS ADR(bDir);
	p_bDirBl ACCESS ADR(bDirBl);
	p_bNoIndexPulse ACCESS ADR(bNoIndexPulse);
	p_usiNode ACCESS ADR(usiNode);
	p_sDevice ACCESS ADR(sDevice);
	p_sProgNm ACCESS ADR(sProgNm);
	p_diMoveBacklashDistInUM ACCESS ADR(diMoveBacklashDistInUM);
	p_diPitchInUM ACCESS ADR(diPitchInUM);
	p_tyParamInHm ACCESS ADR(tyParamInHm);
	p_tyParamInConvert ACCESS ADR(tyParamInConvert);
	p_bNtSettingsLoadDone ACCESS ADR(bNtSettingsLoadDone);
	p_eNtParamMotorType ACCESS ADR(eMotorType);

END_ACTION
```

#### Act_Initial.st - Do Not Change!!!
```iecst
(** 2020-03-16 **)
ACTION Act_Initial:

	//Initial
	sStatTxt	:= a_sStatText[eStat];

	tyParamInMove.diBacklashDistInUM	:= p_diMoveBacklashDistInUM;
	tyParamInMove.diAcc					:= p_diMoveAcc;
	tyParamInMove.diDec					:= p_diMoveDec;

	//p_tyParamInConvert.diPitchInUM	:= fPitchCalc(p_diWidthOffsetInUM , p_diMaxWidthInUM , p_diMinWidthInUM , p_diPitchInUM);

	fbModuleOK.sDevice	:= p_sDevice;
	fbModuleOK.usiNode	:= p_usiNode;
	fbModuleOK.tDlyTm	:= T#5s;
	fbModuleOK(bEn := FALSE);

	fbSDOWrite.sDevice	:= p_sDevice;
	fbSDOWrite.usiNode	:= p_usiNode;
	fbSDOWrite.eMotorType	:= p_eNtParamMotorType;
	fbSDOWrite(bEn := FALSE);

	fbFullMovAbsBl.p_tyParamOutDriver				:= ADR(tyParamOutDriver);
	fbFullMovAbsBl.tyParamInMove.diBacklashDistInUM	:= p_diMoveBacklashDistInUM;
	fbFullMovAbsBl.tyParamInMove.diAcc				:= p_diMoveAcc;
	fbFullMovAbsBl.tyParamInMove.diDec				:= p_diMoveDec;
	//fbFullMovAbsBl.tyParamInConvert					:= p_tyParamInConvert;
	fbFullMovAbsBl.bDir								:= p_bDir;
	fbFullMovAbsBl.bDirBl							:= p_bDirBl;
	fbFullMovAbsBl.bNoIndexPulse					:= p_bNoIndexPulse;
	fbFullMovAbsBl.eMotorType						:= p_eNtParamMotorType;
	fbFullMovAbsBl(bEn := FALSE);

	fbFullMovAbs.p_tyParamOutDriver					:= ADR(tyParamOutDriver);
	fbFullMovAbs.tyParamInMove.diBacklashDistInUM	:= p_diMoveBacklashDistInUM;
	fbFullMovAbs.tyParamInMove.diAcc				:= p_diMoveAcc;
	fbFullMovAbs.tyParamInMove.diDec				:= p_diMoveDec;
	fbFullMovAbs.tyParamInConvert					:= p_tyParamInConvert;
	fbFullMovAbs.bDir								:= p_bDir;
	fbFullMovAbs.bNoIndexPulse						:= p_bNoIndexPulse;
	fbFullMovAbs.eMotorType							:= p_eNtParamMotorType;
	fbFullMovAbs(bEn := FALSE);

	fbFullHm.p_tyParamOutDriver	:= ADR(tyParamOutDriver);
	fbFullHm.bDir				:= p_bDir;
	fbFullHm.bNoIndexPulse		:= p_bNoIndexPulse;
	fbFullHm.eMotorType			:= p_eNtParamMotorType;
	fbFullHm(bEn := FALSE);

	fbPwrOn.p_tyParamOutDriver	:= ADR(tyParamOutDriver);
	fbPwrOn.eMotorType			:= p_eNtParamMotorType;
	fbPwrOn(bEn := FALSE);

	fbPwrOff.p_tyParamOutDriver	:= ADR(tyParamOutDriver);
	fbPwrOff.eMotorType			:= p_eNtParamMotorType;
	fbPwrOff(bEn := FALSE);

	fbHoming.p_tyParamOutDriver	:= ADR(tyParamOutDriver);
	fbHoming.bDir				:= p_bDir;
	fbHoming.bNoIndexPulse		:= p_bNoIndexPulse;
	fbHoming.eMotorType			:= p_eNtParamMotorType;
	fbHoming(bEn := FALSE);

	fbMovAbs.p_tyParamOutDriver					:= ADR(tyParamOutDriver);
	fbMovAbs.tyParamInMove.diBacklashDistInUM	:= p_diMoveBacklashDistInUM;
	fbMovAbs.tyParamInMove.diAcc				:= p_diMoveAcc;
	fbMovAbs.tyParamInMove.diDec				:= p_diMoveDec;
	fbMovAbs.tyParamInConvert					:= p_tyParamInConvert;
	fbMovAbs.bDir								:= p_bDir;
	fbMovAbs.eMotorType							:= p_eNtParamMotorType;
	fbMovAbs(bEn := FALSE);

	fbMovRel.p_tyParamOutDriver					:= ADR(tyParamOutDriver);
	fbMovRel.tyParamInMove.diBacklashDistInUM	:= p_diMoveBacklashDistInUM;
	fbMovRel.tyParamInMove.diAcc				:= p_diMoveAcc;
	fbMovRel.tyParamInMove.diDec				:= p_diMoveDec;
	fbMovRel.tyParamInConvert					:= p_tyParamInConvert;
	fbMovRel.bDir								:= p_bDir;
	fbMovRel.eMotorType							:= p_eNtParamMotorType;
	fbMovRel(bEn := FALSE);

	fbJog.p_tyParamOutDriver	:= ADR(tyParamOutDriver);
	fbJog.tyParamInConvert		:= p_tyParamInConvert;
	fbJog.eMotorType			:= p_eNtParamMotorType;
	fbJog(bEn := FALSE);

	fbRstAxisErr.p_tyParamOutDriver	:= ADR(tyParamOutDriver);
	fbRstAxisErr(bEn := FALSE);

	fbStop.p_tyParamOutDriver	:= ADR(tyParamOutDriver);
	fbStop(bEn := FALSE);

	bModuleNotOK	:= TRUE;

END_ACTION
```

#### Act_Background.st - Do Not Change!!!
```iecst
(** 2020-05-26 **)
ACTION Act_Background:

	//Update Parameter
	IF bModuleOK = TRUE THEN

		tyParamInMove.diPosInUM		:= p_diMovePosInUM;
		tyParamInMove.diDistInUM	:= p_diMoveDistInUM;
		tyParamInMove.diVelInUMPS	:= p_diMoveVelInUMPS;
		tyParamInMove.diAcc			:= p_diMoveAcc;
		tyParamInMove.diDec			:= p_diMoveDec;

		fMotionCANUpdtDat(ADR(tyParamOut) , p_tyParamInConvert , tyParamOutDriver , tyParamInDriver , tyParamInMove , p_tyParamInHm , p_bDir, p_eNtParamMotorType);

		bWidthPosDiff	:= (tyParamOut.bIsHomed = FALSE) OR ((ABS((fAWWidthToPosInUM(p_diGoWidth , p_diWidthAtHmPos)) - tyParamOut.diActualPosInUM)) > 500);

		p_tyParamInConvert.diPitchInUM	:= fPitchCalc(p_diWidthOffsetInUM , p_diMaxWidthInUM , p_diMinWidthInUM , p_diPitchInUM);

		fbFullMovAbsBl.tyParamInConvert					:= p_tyParamInConvert;

		IF p_bDir = TRUE THEN
			bOpenSen	:= tyParamOut.bFwdLmtSen;
			bCloseSen	:= tyParamOut.bRevLmtSen;
		ELSE
			bOpenSen	:= tyParamOut.bRevLmtSen;
			bCloseSen	:= tyParamOut.bFwdLmtSen;
		END_IF

		CASE p_eNtParamMotorType OF
			DeltaAsdaA2:
				CASE tyParamOut.udiAxisErrID OF
					8976:	sAxisErrTxt	:= 'Over Current';
					12560:	sAxisErrTxt	:= 'Over Voltage';
					12576:	sAxisErrTxt	:= 'Under Voltage';
					12592:	sAxisErrTxt	:= 'Input Power Phase Loss';
					12816:	sAxisErrTxt	:= 'Regeneration Error';
					12848:	sAxisErrTxt	:= 'Overload';
					12849:	sAxisErrTxt	:= 'Pre-overload Warning';
					13056:	sAxisErrTxt	:= 'U,V,W Wiring Error';
					16912:	sAxisErrTxt	:= 'IGBT Temperature Error';
					21296:	sAxisErrTxt	:= 'Memory Error';
					21569:	sAxisErrTxt	:= 'Emergency Stop Activated';
					21570:	sAxisErrTxt	:= 'Forward Limit Switch Error';
					21571:	sAxisErrTxt	:= 'Reverse Limit Switch Error';
					21572:	sAxisErrTxt	:= 'Forward Software Limit';
					21573:	sAxisErrTxt	:= 'Reverse Software Limit';
					21760:	sAxisErrTxt	:= 'DSP Firmware Upgrade';
					25088:	sAxisErrTxt	:= 'CANopen SYNC Error';
					25360:	sAxisErrTxt	:= 'CANopen Data Initial Error';
					25376:	sAxisErrTxt	:= 'Adjustment Error';
					28961:	sAxisErrTxt	:= 'Motor Protection Error';
					28962:	sAxisErrTxt	:= 'Motor Error';
					29445:	sAxisErrTxt	:= 'Encoder Error';
					29446:	sAxisErrTxt	:= 'Encoder Output Error';
					29968:	sAxisErrTxt	:= 'Serial Communication Error';
					29984:	sAxisErrTxt	:= 'Serial Communication Time Out';
					33024:	sAxisErrTxt	:= 'CANbus Error (Bus-off)';
					33040:	sAxisErrTxt	:= 'CANopen SDO receive buffer overrun';
					33056:	sAxisErrTxt	:= 'CANbus Error (Warning)';
					33072:	sAxisErrTxt	:= 'Node Guarding or Heartbeat Error';
					33280:	sAxisErrTxt	:= 'CANopen PDO Object Error';
					33792:	sAxisErrTxt	:= 'Over Speed';
					34304:	sAxisErrTxt	:= 'Abnormal Pulse Control Command';
					34320:	sAxisErrTxt	:= 'Full Closed Loop Excessive Deviation';
					34321:	sAxisErrTxt	:= 'Excessive Deviation';
				END_CASE

			SchneiderLexium28:
				CASE tyParamOut.udiAxisErrID OF
					8724:	sAxisErrTxt	:= 'Over Current';
					8976:	sAxisErrTxt	:= 'Motor Overload';
					8977:	sAxisErrTxt	:= 'Drive overload (foldback)';
					9088:	sAxisErrTxt	:= 'Calculated offsets for current sensors out OF range';
					9089:	sAxisErrTxt := 'Motor phase missing';
					9090:	sAxisErrTxt := 'Overcurrent detected at one OF the digital outputs';
					12560:	sAxisErrTxt	:= 'DC Bus Over Voltage';
					12576:	sAxisErrTxt	:= 'DC Bus Under Voltage';
					12672:	sAxisErrTxt	:= 'Braking Resistor Overload';
					12673:	sAxisErrTxt	:= 'Safety function Safe Torque Off (STO) triggered';
					12674:	sAxisErrTxt	:= 'DC bus voltage measurement';
					12675:	sAxisErrTxt	:= 'Missing mains supply, undervoltage mains supply';
					12676:	sAxisErrTxt := 'The encoder supply voltage has dropped under operational value';
					12677:	sAxisErrTxt := 'The multi turn encoder battery voltage has dropped under 3 Vdc';
					12678:	sAxisErrTxt := 'Internal position synchronization error	detected between the multi turn AND the single turn modules';
					12679:	sAxisErrTxt := 'Generic error code of the multi turn module is detected';
					12697:	sAxisErrTxt := 'Braking resistor overload';
					16512:	sAxisErrTxt	:= 'Drive overtemperature (IPM)';
					16513:	sAxisErrTxt	:= 'Drive overtemperature (controller)';
					16534:	sAxisErrTxt := 'Temperature sensor inoperative';
					17168:	sAxisErrTxt	:= 'Power stage overtemperature';
					17280:	sAxisErrTxt := 'The encoder temperature is too high';
					17424:	sAxisErrTxt	:= 'Motor overtemperature';
					21808:	sAxisErrTxt	:= 'System error detected (nonvolatilememory)';
					21893:	sAxisErrTxt	:= 'Error detected in non-volatile memory';
					21889:	sAxisErrTxt	:= 'System error detected (nonvolatile memory)';
					21890:	sAxisErrTxt	:= 'System error detected (CAN power supply)';
					21891:	sAxisErrTxt	:= 'System error detected (selftest)';
					21894:	sAxisErrTxt	:= 'System error detected (NV ACCESS)';
					25472:	sAxisErrTxt	:= 'Target position rejected';
					25985:	sAxisErrTxt	:= 'System error detected(FPGA)';
					28816:	sAxisErrTxt	:= 'System error detected (FPGA does NOT match firmware)';
					28817:	sAxisErrTxt	:= 'Emergency Stop Activated';
					28961:	sAxisErrTxt := 'Motor blocked';
					29080:	sAxisErrTxt := 'Commutation error detected';
					29568:  sAxisErrTxt	:= 'Error detected in communication with motor encoder';
					29574:	sAxisErrTxt	:= 'Drive is not synchronous wit master cycle';
					29581:	sAxisErrTxt := 'System error detected (encoder)';
					29587:	sAxisErrTxt	:= 'Encoder overvoltage or overcurrent';
					29592:	sAxisErrTxt := 'The returned position value are no longer considered valid';
					29593:	sAxisErrTxt := 'The multi turn encoder requires an explicit configuration command';
					30081:	sAxisErrTxt := 'Target position rejected';
					30082:	sAxisErrTxt := 'No target values received via the fieldbus';
					33072:	sAxisErrTxt	:= 'CANopen: Heartbeat error detected';
					33296:	sAxisErrTxt := 'R_PDO is too short';
					33921:	sAxisErrTxt	:= 'Actual Motor Velocity Too High';
					33553:	sAxisErrTxt	:= 'Motor torque too high FOR an excessive period OF time';
					33664:	sAxisErrTxt := 'Unstable current loop';
					33922:	sAxisErrTxt := 'Velocity deviation too high';
					34321:	sAxisErrTxt	:= 'Position deviation too high';
					34432:	sAxisErrTxt := 'Position deviation via signal output function MC_OK';
					34441:	sAxisErrTxt := 'Position deviation too high (following error)';
					61568:	sAxisErrTxt	:= 'Fieldbus: Communication	error detected';
					65282:	sAxisErrTxt	:= 'Not possible to read data of electronic motor nameplate';
					65296:	sAxisErrTxt	:= 'Forward Limit Switch Error';
					65297:	sAxisErrTxt	:= 'Reverse Limit Switch Error';
					65281:	sAxisErrTxt := 'System error detected';
					65298:	sAxisErrTxt	:= 'Forward Software Limit';
					65299:	sAxisErrTxt	:= 'Reverse Software Limit';
					65301:	sAxisErrTxt := 'The encoder firmware cannot operate on the provided hardware';

				END_CASE

			EstunPronet:
				CASE tyParamOut.udiAxisErrID OF
					65281:	sAxisErrTxt	:= 'Parameter breakdown';//A01
					65282:	sAxisErrTxt	:= 'AD shift channels breakdown';
					65283:	sAxisErrTxt	:= 'Overspeed';
					65284:	sAxisErrTxt	:= 'Overload';
					65285:	sAxisErrTxt := 'Position error counteroverflow ';
					65286:	sAxisErrTxt := 'Position error pulse overflow';
					65287:	sAxisErrTxt	:= 'The setting of electronic gear or given pulse frequency is not reasonable';
					65288:	sAxisErrTxt	:= 'The 1st channel of current detection is wrong.';
					65289:	sAxisErrTxt	:= 'The 2nd channel of current detection is wrong.';
					65290:	sAxisErrTxt	:= 'Incremental Encoder is break off.';//A10
					65292:	sAxisErrTxt	:= 'Overcurrent';
					65293:	sAxisErrTxt	:= 'Overvoltage';
					65294:	sAxisErrTxt	:= 'Undervoltage';
					65295:	sAxisErrTxt := 'Bleeder resistor error';
					65296:	sAxisErrTxt := 'Regeneration error';
					65297:	sAxisErrTxt := 'Resolver error';
					65298:	sAxisErrTxt := 'IGBT superheat alarm';
					65299:	sAxisErrTxt := 'Motor overheat alarm';
					65300:	sAxisErrTxt := 'Power line phase shortage';//A20
					65301:	sAxisErrTxt	:= 'Instantaneous power off alarm';
					65302:	sAxisErrTxt	:= 'Motor temperature detection sensor is break off.';
					65303:	sAxisErrTxt := 'Brake overcurrent alarm';//A23
					65305:	sAxisErrTxt := 'Motor power line U overcurrent';//A25
					65306:	sAxisErrTxt := 'Motor power line V overcurrent';//A26
					65307:	sAxisErrTxt := 'Motor power line W overcurrent';//A27
					65322:	sAxisErrTxt	:= 'Servomotor type error';//A42
					65323:	sAxisErrTxt	:= 'Servo drive type error';
					65325:	sAxisErrTxt	:= 'Absolute encoder multiturn information error';
					65326:	sAxisErrTxt	:= 'Absolute encoder multiturn information overflow';
					65327:	sAxisErrTxt	:= 'Battery voltage below 2.5V';
					65328:	sAxisErrTxt	:= 'Battery voltage below 3.1V';//A48
					65330:	sAxisErrTxt := 'Serial encoder communication overtime ';//A50
					65331:	sAxisErrTxt := 'Absolute encoder overspeed alarm detected';
					65332:  sAxisErrTxt	:= 'Absolute state of serial encoder error';
					65333:	sAxisErrTxt	:= 'Serial encoder calcaution error';
					65334:	sAxisErrTxt := 'Parity bit or end bit in serial encoder control domain error';
					65335:	sAxisErrTxt	:= 'Serial encoder communication data checking error';
					65336:	sAxisErrTxt := 'End bit in serial encoder control domain error';
					65338:	sAxisErrTxt := 'Serial encoder data empty';
					65339:	sAxisErrTxt := 'Serial encoder data format error';
					65340:	sAxisErrTxt := 'Communication module not detected ';//A60
					65341:	sAxisErrTxt := 'Communication unsuccessful';
					65342:	sAxisErrTxt := 'Servo drive can not receive the period data of communication module ';
					65343:	sAxisErrTxt := 'Communication module can not receive the servo drive response data.';
					65344:	sAxisErrTxt := 'Communication module and bus connectionless';
					65346:	sAxisErrTxt := 'CAN communication abnormal';
					65347:	sAxisErrTxt := 'Receiving heartbeat timeout';
					65349:	sAxisErrTxt := 'Synchronization signal monitoring cycle is longer than setting';
					65362: sAxisErrTxt	:= 'Torque output alarm';
				END_CASE
		END_CASE

	ELSE

		tyParamOut.bAxisErr			:= FALSE;
		tyParamOut.bFwdLmtSen		:= FALSE;
		tyParamOut.bInPos			:= FALSE;
		tyParamOut.bIsHomed			:= FALSE;
		tyParamOut.bPosDiff			:= TRUE;
		tyParamOut.bPwrOn			:= FALSE;
		tyParamOut.bRevLmtSen		:= FALSE;
		tyParamOut.bStopped			:= TRUE;
		tyParamOut.diActualPosInUM	:= 0;
		tyParamOut.diHmAcc			:= 0;
		tyParamOut.diHmSpdForSwitch	:= 0;
		tyParamOut.diHmSpdForZero	:= 0;
		tyParamOut.diProfileAcc		:= 0;
		tyParamOut.diProfileDec		:= 0;
		tyParamOut.udiAxisErrID		:= 0;

		bWidthPosDiff				:= TRUE;

	END_IF

	//Abnormal Movement
	IF eStatus1 <> Error THEN
		IF p_bOps = TRUE AND eStatus = Idle THEN
			IF (ABS(tyParamOut.diActualPosInUM - diActualPosInUMOld) > 2000) AND (ABS(tyParamOut.diActualPosInUM - diActualPosInUMOld) < 10000) THEN
				eStatus1	:= Error;
				udiStatus1	:= 10000;	//Axis Move Abnormally By External Force

				fMotionCANRstCtrlWord(ADR(tyParamOutDriver));
				p_eAct	:= AWActIdle;
				eStat	:= AWActIdle;
			END_IF
		ELSE
			diActualPosInUMOld	:= tyParamOut.diActualPosInUM;
		END_IF
	END_IF

	//Reset Error
	IF (eStatus1 = Error) AND bRstErr THEN
		eStatus1	:= Idle;
		udiStatus1	:= 0;
	END_IF

	//Request Position To Movement Out Of Range
	IF p_bOps
		AND((tyParamInMove.diPosInUM < p_diMinAbsPosInUM) OR (tyParamInMove.diPosInUM > p_diMaxAbsPosInUM))
		AND (eStatus2 <> Error) THEN
		eStatus2	:= Error;
		udiStatus2	:= 10029;	//Request Absolute Position Out Of Range

		fMotionCANRstCtrlWord(ADR(tyParamOutDriver));
		p_eAct	:= AWActIdle;
		eStat	:= AWActIdle;
	END_IF

	//Reset Error
	IF (eStatus2 = Error) AND bRstErr THEN
		eStatus2	:= Idle;
		udiStatus2	:= 0;
	END_IF

	//Sensor Interrupt
	IF (bNotInterruptible = TRUE OR bJogging) AND eStatus3 <> Error THEN

		IF p_bInletSensor = TRUE THEN
			eStatus3	:= Error;
			udiStatus3	:= 10030;	//Inlet Sensor Interrupt Auto Width Movement

			fMotionCANRstCtrlWord(ADR(tyParamOutDriver));
			p_eAct	:= AWActIdle;
			eStat	:= AWActIdle;

		ELSIF p_bOutletSensor = TRUE THEN
			eStatus3	:= Error;
			udiStatus3	:= 10031;	//Outlet Sensor Interrupt Auto Width Movement

			fMotionCANRstCtrlWord(ADR(tyParamOutDriver));
			p_eAct	:= AWActIdle;
			eStat	:= AWActIdle;

		ELSIF p_bClearSensor = TRUE THEN
			eStatus3	:= Error;
			udiStatus3	:= 10032;	//Clear Sensor Interrupt Auto Width Movement

			fMotionCANRstCtrlWord(ADR(tyParamOutDriver));
			p_eAct	:= AWActIdle;
			eStat	:= AWActIdle;

		ELSIF p_bMiddleSensor = TRUE THEN
			eStatus3	:= Error;
			udiStatus3	:= 10033;	//Middle Sensor Interrupt Auto Width Movement

			fMotionCANRstCtrlWord(ADR(tyParamOutDriver));
			p_eAct	:= AWActIdle;
			eStat	:= AWActIdle;

		ELSIF p_bInterruptSensor = TRUE THEN
			eStatus3	:= Error;
			udiStatus3	:= 10034;	//Sensor Interrupt Auto Width Movement

			fMotionCANRstCtrlWord(ADR(tyParamOutDriver));
			p_eAct	:= AWActIdle;
			eStat	:= AWActIdle;

		ELSIF p_bCloseInterruptSensor = TRUE AND bJogOpen = FALSE THEN
			eStatus3	:= Error;
			udiStatus3	:= 10047;	//Sensor Interrupt Auto Width Movement

			fMotionCANRstCtrlWord(ADR(tyParamOutDriver));
			p_eAct	:= AWActIdle;
			eStat	:= AWActIdle;

		ELSIF p_bOpenInterruptSensor = TRUE AND bJogClose = FALSE THEN
			eStatus3	:= Error;
			udiStatus3	:= 10048;	//Sensor Interrupt Auto Width Movement

			fMotionCANRstCtrlWord(ADR(tyParamOutDriver));
			p_eAct	:= AWActIdle;
			eStat	:= AWActIdle;
		END_IF

	END_IF

	//Reset Error
	IF (eStatus3 = Error AND bRstErr)
		OR (p_bOpenInterruptSensor AND eStat = AWActJogClose)
		OR (p_bCloseInterruptSensor AND eStat = AWActJogOpen)
		THEN
		eStatus3	:= Idle;
		udiStatus3	:= 0;
	END_IF

	IF bRstErr THEN
		udiStatus	:= 0;
		bJogging	:= FALSE;
		bJogClose	:= FALSE;
		bJogOpen	:= FALSE;
	END_IF

	fbServoModuleOk(IN:= bModuleOK);
	fbServoModuleNotOk(IN:= bModuleOK = FALSE);
	IF fbServoModuleNotOk.Q AND udiStatus <> 10001 THEN

		bModuleNotOK		:= TRUE;
		bModuleNotOKLock	:= TRUE;
		usiRstStep	:= 0;
		tyParamOutDriver.uiCtrlword_6040	:= 0;
		tyParamOutDriver.siModOfOpt_6060	:= 0;
		tyParamOutDriver.diTargetPos_607A	:= 0;
		tyParamOutDriver.udiMoveSpd_6081	:= 0;
		tyParamOutDriver.siHmMethod_6098	:= 0;
		tyParamOutDriver.diJogVel_60FF		:= 0;

		CASE p_eNtParamMotorType OF

			DeltaAsdaA2:
				fbModuleOK(bModuleOK:= FALSE);
				IF eStatus = Idle THEN
					eAct	:= AWActRstNode;
				END_IF

				IF (eStatus = Done OR eStatus = Error)AND eStat = AWActRstNode THEN

					eAct	:= AWActIdle;
				END_IF

			EstunPronet:
				fbModuleOK(bModuleOK:= FALSE);
				IF eStatus = Idle THEN
					eAct	:= AWActRstNode;
				END_IF

				IF (eStatus = Done OR eStatus = Error)AND eStat = AWActRstNode THEN

					eAct	:= AWActIdle;
				END_IF

			SchneiderLexium28:
			// Do Nothing
		END_CASE

	ELSIF bModuleNotOK = TRUE AND fbServoModuleOk.Q THEN

		CASE usiRstStep OF

			0:
				IF eStatus = Idle THEN
					eAct	:= AWActRstAxisErr;
				END_IF

				IF eStatus = Done AND eStat = AWActRstAxisErr THEN
					eAct	:= AWActIdle;
					usiRstStep	:= 4;
				END_IF

			4: tyParamOutDriver.siModOfOpt_6060 := 1;
				usiRstStep	:= 5;

			5: tyParamOutDriver.siModOfOpt_6060 := 1;
				fbRstNodeTimer(IN:=TRUE);

				IF tyParamInDriver.siModOfOptDisp_6061 = 1 THEN
					usiRstStep	:= 6;
					fbRstNodeTimer(IN:=FALSE);
				ELSIF fbRstNodeTimer.Q THEN
					usiRstStep	:= 8;
					fbRstNodeTimer(IN:=FALSE);
				END_IF

			6: tyParamOutDriver.siModOfOpt_6060 := 6;
				fbRstNodeTimer(IN:=FALSE);
				usiRstStep	:= 7;

			7: tyParamOutDriver.siModOfOpt_6060 := 6;
				fbRstNodeTimer(IN:=TRUE);

				IF tyParamInDriver.siModOfOptDisp_6061 = 6 THEN
					usiRstStep	:= 10;
					fbRstNodeTimer(IN:=FALSE);
				ELSIF fbRstNodeTimer.Q THEN
					usiRstStep	:= 9;
					fbRstNodeTimer(IN:=FALSE);
				END_IF

			8:	fbModuleOK(bEn := TRUE, bModuleOK:= FALSE);
				fbRstNodeTimer(IN:=FALSE);
				usiRstStep	:= 9;

			9:	fbModuleOK(bModuleOK:= FALSE);
				IF eStatus = Idle THEN
					eAct	:=AWActRstNode;
				END_IF

				IF eStatus = Done AND eStat = AWActRstNode THEN
					usiRstStep	:= 0;
					eAct		:= AWActIdle;
				END_IF

			10:IF eStatus = Idle THEN
					eAct	:= AWActRstAxisErr;
				END_IF

				IF eStatus = Done AND eStat = AWActRstAxisErr THEN
					eAct			:=AWActIdle;
					usiRstStep	:= 11;
				END_IF

			11:

				IF eStatus = Idle THEN
					eAct	:= AWActSDOWrite;
				END_IF

				IF eStatus = Done AND eStat = AWActSDOWrite THEN
					eAct			:= AWActIdle;
					usiRstStep	:= 13;

				ELSIF udiStatus = 10028 THEN
					eAct			:= AWActIdle;
					usiRstStep	:= 0;
				END_IF

			13: bModuleNotOK	:= FALSE;
				usiRstStep	:= 0;
		END_CASE
	ELSE
		eAct	:= AWActIdle;

	END_IF

	IF tyParamOut.bPosDiff = FALSE THEN
		tyParamOutDriver.uiCtrlword_6040.4	:= FALSE;
	END_IF

END_ACTION
```

#### Act_Alarm.st - Do Not Change!!!
```iecst
(** 2020-03-16 **)
ACTION Act_Alarm:

	//Error
	IF EDGEPOS(eStatus = Error) THEN

		tyAlmData.sProgNm		:= p_sProgNm;
		tyAlmData.udiCode		:= udiStatus;
		tyAlmData.eSeverity		:= AlmSeverityError;
		tyAlmData.udiRunTime	:= tyAlmData.udiRunTime + 1;
		tyAlmData.bAlm			:= TRUE;
		tyAlmData.udiModuleNum  := udiModuleNum;
		g_sAWOpenProgNm			:= p_sProgNm;

		//Get Error Message
		IF tyAlmData.udiCode < 10000 OR tyAlmData.udiCode > 10299 THEN
			tyAlmData.sAlmMsg	:= 'Unknown';
			tyAlmData.sRcyMsg	:= 'Unknown';
		ELSE
			tyAlmData.sAlmMsg	:= a_tyAlmText[tyAlmData.udiCode].sAlmText;
			tyAlmData.sRcyMsg	:= a_tyAlmText[tyAlmData.udiCode].sRcyText;
		END_IF

		sStatTxt	:= tyAlmData.sAlmMsg;

	ELSIF bRstErr AND (tyAlmData.udiCode <> 0) THEN

		tyAlmData.udiCode	:= 0;
		tyAlmData.eSeverity	:= AlmSeverityNA;
		tyAlmData.sAlmMsg	:= '';
		tyAlmData.sRcyMsg	:= '';
		tyAlmData.bAlm			:= FALSE;
		sStatTxt	:= a_sStatText[eStat];

	END_IF

END_ACTION
```

#### Act_Alarm1.st - Do Not Change!!!
```iecst
(** 2020-03-16 **)
ACTION Act_Alarm1:

	//Error
	IF EDGEPOS(eStatus1 = Error) THEN

		tyAlmData1.sProgNm		:= p_sProgNm;
		tyAlmData1.udiCode		:= udiStatus1;
		tyAlmData1.eSeverity	:= AlmSeverityError;
		tyAlmData1.udiRunTime	:= tyAlmData1.udiRunTime + 1;
		tyAlmData1.bAlm			:= TRUE;
		tyAlmData1.udiModuleNum  := udiModuleNum;
		g_sAWOpenProgNm		:= p_sProgNm;
		//Get Error Message
		IF tyAlmData1.udiCode < 10000 OR tyAlmData1.udiCode > 10099 THEN
			tyAlmData1.sAlmMsg	:= 'Unknown';
			tyAlmData1.sRcyMsg	:= 'Unknown';
		ELSE
			tyAlmData1.sAlmMsg	:= a_tyAlmText[tyAlmData1.udiCode].sAlmText;
			tyAlmData1.sRcyMsg	:= a_tyAlmText[tyAlmData1.udiCode].sRcyText;
		END_IF

		sStatTxt	:= tyAlmData1.sAlmMsg;

	ELSIF bRstErr AND (tyAlmData1.udiCode <> 0) THEN

		tyAlmData1.udiCode		:= 0;
		tyAlmData1.eSeverity	:= AlmSeverityNA;
		tyAlmData1.sAlmMsg		:= '';
		tyAlmData1.sRcyMsg		:= '';
		tyAlmData1.bAlm			:= FALSE;
		sStatTxt	:= a_sStatText[eStat];

	END_IF

END_ACTION
```

#### Act_Alarm2.st - Do Not Change!!!
```iecst
(** 2020-03-16 **)
ACTION Act_Alarm2:

	//Error
	IF EDGEPOS(eStatus2 = Error) THEN

		tyAlmData2.sProgNm		:= p_sProgNm;
		tyAlmData2.udiCode		:= udiStatus2;
		tyAlmData2.eSeverity	:= AlmSeverityError;
		tyAlmData2.udiRunTime	:= tyAlmData2.udiRunTime + 1;
		tyAlmData2.bAlm			:= TRUE;
		tyAlmData2.udiModuleNum  := udiModuleNum;
		g_sAWOpenProgNm		:= p_sProgNm;
		//Get Error Message
		IF tyAlmData2.udiCode < 10000 OR tyAlmData2.udiCode > 10099 THEN
			tyAlmData2.sAlmMsg	:= 'Unknown';
			tyAlmData2.sRcyMsg	:= 'Unknown';
		ELSE
			tyAlmData2.sAlmMsg	:= a_tyAlmText[tyAlmData2.udiCode].sAlmText;
			tyAlmData2.sRcyMsg	:= a_tyAlmText[tyAlmData2.udiCode].sRcyText;
		END_IF

		sStatTxt	:= tyAlmData2.sAlmMsg;

	ELSIF bRstErr AND (tyAlmData2.udiCode <> 0) THEN

		tyAlmData2.udiCode		:= 0;
		tyAlmData2.eSeverity	:= AlmSeverityNA;
		tyAlmData2.sAlmMsg		:= '';
		tyAlmData2.sRcyMsg		:= '';
		tyAlmData2.bAlm			:= FALSE;
		sStatTxt	:= a_sStatText[eStat];

	END_IF

END_ACTION
```

#### Act_Alarm3.st - Do Not Change!!!
```iecst
(** 2020-03-16 **)
ACTION Act_Alarm3:

	//Error
	IF EDGEPOS(eStatus3 = Error) THEN

		tyAlmData3.sProgNm		:= p_sProgNm;
		tyAlmData3.udiCode		:= udiStatus3;
		tyAlmData3.eSeverity	:= AlmSeverityError;
		tyAlmData3.udiRunTime	:= tyAlmData3.udiRunTime + 1;
		tyAlmData3.bAlm			:= TRUE;
		tyAlmData3.udiModuleNum  := udiModuleNum;
		g_sAWOpenProgNm		:= p_sProgNm;
		//Get Error Message
		IF tyAlmData3.udiCode < 10000 OR tyAlmData3.udiCode > 10099 THEN
			tyAlmData3.sAlmMsg	:= 'Unknown';
			tyAlmData3.sRcyMsg	:= 'Unknown';
		ELSE
			tyAlmData3.sAlmMsg	:= a_tyAlmText[tyAlmData3.udiCode].sAlmText;
			tyAlmData3.sRcyMsg	:= a_tyAlmText[tyAlmData3.udiCode].sRcyText;
		END_IF

		sStatTxt	:= tyAlmData3.sAlmMsg;

	ELSIF bRstErr AND (tyAlmData3.udiCode <> 0) THEN

		tyAlmData3.udiCode		:= 0;
		tyAlmData3.eSeverity	:= AlmSeverityNA;
		tyAlmData3.sAlmMsg		:= '';
		tyAlmData3.sRcyMsg		:= '';
		tyAlmData3.bAlm			:= FALSE;
		sStatTxt	:= a_sStatText[eStat];

	END_IF

END_ACTION
```

#### InputRef.var - Do Not Change!!!
```iecst
(*2020-05-26*)
(**)
(*General*)
VAR
	p_eAct : REFERENCE TO eAWAction;
	p_udiRstErr : REFERENCE TO UDINT;
	p_bPrep : REFERENCE TO BOOL;
	p_bEn : REFERENCE TO BOOL;
	p_bDis : REFERENCE TO BOOL;
END_VAR
(**)
(*Configuration*)
VAR
	p_bOps : REFERENCE TO BOOL;
	p_bManual : REFERENCE TO BOOL;
	p_diWidthAtHmPos : REFERENCE TO DINT;
	p_tyTuning : REFERENCE TO tyMotionCANTuning;
	p_diGoWidth : REFERENCE TO DINT;
	p_diJogVelInUMPS : REFERENCE TO DINT;
	p_diMovePosInUM : REFERENCE TO DINT;
	p_diMoveDistInUM : REFERENCE TO DINT;
	p_diMoveVelInUMPS : REFERENCE TO DINT;
	p_diMoveAcc : REFERENCE TO DINT;
	p_diMoveDec : REFERENCE TO DINT;
	p_diMinAbsPosInUM : REFERENCE TO DINT;
	p_diMaxAbsPosInUM : REFERENCE TO DINT;
	p_diMinWidthInUM : REFERENCE TO DINT;
	p_diMaxWidthInUM : REFERENCE TO DINT;
	p_diWidthOffsetInUM : REFERENCE TO DINT;
	p_bInletSensor : REFERENCE TO BOOL;
	p_bOutletSensor : REFERENCE TO BOOL;
	p_bClearSensor : REFERENCE TO BOOL;
	p_bMiddleSensor : REFERENCE TO BOOL;
	p_bInterruptSensor : REFERENCE TO BOOL;
	p_bOpenInterruptSensor : REFERENCE TO BOOL;
	p_bCloseInterruptSensor : REFERENCE TO BOOL;
	p_bSafetyInterruptSen : REFERENCE TO BOOL;
	p_bDir : REFERENCE TO BOOL;
	p_bDirBl : REFERENCE TO BOOL;
	p_bNoIndexPulse : REFERENCE TO BOOL;
	p_usiNode : REFERENCE TO USINT;
	p_sDevice : REFERENCE TO STRING[3];
	p_sProgNm : REFERENCE TO STRING[15];
	p_diMoveBacklashDistInUM : REFERENCE TO DINT;
	p_diPitchInUM : REFERENCE TO DINT;
	p_tyParamInHm : REFERENCE TO tyMotionCANParamInHm;
	p_tyParamInConvert : REFERENCE TO tyMotionCANParamInConvert;
	p_bNtSettingsLoadDone : REFERENCE TO BOOL;
	p_bOpsAWStepMove : REFERENCE TO BOOL;
	p_eNtParamMotorType : REFERENCE TO eServoMotorType;
	p_bOutletShutterCloseRS : REFERENCE TO BOOL;
	p_bOutletShutterCloseRS3 : REFERENCE TO BOOL;
	p_bOutletShutterCloseRS2 : REFERENCE TO BOOL;
	p_bProjInletShutPrep : REFERENCE TO BOOL;
	p_bInShutterDis : REFERENCE TO BOOL;
	p_bProjOutletShutPrep : REFERENCE TO BOOL;
	p_bInletShutterCloseRS : REFERENCE TO BOOL;
	p_bPusherRetSen : REFERENCE TO BOOL;
	p_bPusherExtSen : REFERENCE TO BOOL;
	p_bNtParamAutoRcpPrep : REFERENCE TO BOOL;
	p_bMcParamAutoRcpDis : REFERENCE TO BOOL;
	p_eNtParamAutoRcpPrecededBy : REFERENCE TO eAutoRcpPreceded;
END_VAR
```

#### Local.var - Do Not Change!!!
```iecst
(*2020-05-26*)
(**)
(*Local Action, State & Status*)
VAR
	eAct : eAWAction := AWActIdle;
	eStat : eAWAction := AWActIdle;
	eMainStatus : eFBStatus := Idle;
	eStatus : eFBStatus := Idle;
	eStatus1 : eFBStatus := Idle;
	eStatus2 : eFBStatus := Idle;
	eStatus3 : eFBStatus := Idle;
	udiStatus : UDINT := 0;
	udiStatus1 : UDINT := 0;
	udiStatus2 : UDINT := 0;
	udiStatus3 : UDINT := 0;
	sStatTxt : STRING[200] := '';
	a_sStatText : ARRAY[0..50] OF STRING[200] := ['Idling','Going Width','Full Homing','Powering On','Powering Off','Homing','Moving Absolute','Moving Relative','Jogging Open','Jogging Close','Jogging Stop','Resetting Axis Error','Stopping','Writing SDO','Background Starting Module OK Check','Background Stopping Module OK Check','Going Width And Power Off','Reset Servo Module Node',33('')];
END_VAR
(**)
(*Local Alarm*)
VAR
	tyAlmData : tyAlmDat;
	tyAlmData1 : tyAlmDat;
	tyAlmData2 : tyAlmDat;
	tyAlmData3 : tyAlmDat;
	a_tyAlmText : ARRAY[10000..10299] OF tyAlmTxt := [(sAlmText:='Axis Move Abnormally By External Force',sRcyText:='Servo Motor Abnormal Operation. Reset And Resume Operation. If The Problem Persists, Please Contact Nutek For A Possible Solution.'),(sAlmText:='CANOpen Communication Error, ModuleOK Not TRUE',sRcyText:='Fail While Read/Write Data. Reset The Error And Resume Operation.'),(sAlmText:='Power On Time Out While Going New Width',sRcyText:='Timeout Expired Before Operation Completed. Reset And Resume Operation.'),(sAlmText:='Homing Time Out While Going New Width',sRcyText:='Timeout Expired Before Operation Completed. Reset And Resume Operation.'),(sAlmText:='Move Absolute Time Out While Going New Width',sRcyText:='Timeout Expired Before Operation Completed. Reset And Resume Operation.'),(sAlmText:='Stop Motion Time Out While Going New Width',sRcyText:='Timeout Expired Before Operation Completed. Reset And Resume Operation.'),(sAlmText:='Axis Error Reset Failed While Going New Width',sRcyText:='Axis Error Reset Failed. Please Retry Again Reset Operation. If The Problem Persists, Please Contact Nutek For A Possible Solution.'),(sAlmText:='Axis Error Occur In Move Absolute While Going New Width',sRcyText:='Servo Motor Abnormal Operation. Reset And Resume Operation. If The Problem Persists, Please Contact Nutek For A Possible Solution.'),(sAlmText:='Axis Error Occur In Homing While Going New Width',sRcyText:='Servo Motor Abnormal Operation. Reset And Resume Operation. If The Problem Persists, Please Contact Nutek For A Possible Solution.'),(sAlmText:='Homing Done But Home Flag Is Not Activated While Going New Width',sRcyText:='Servo Motor Abnormal Operation. Reset And Resume Operation. If The Problem Persists, Please Contact Nutek For A Possible Solution.'),(sAlmText:='Forward Limit Activated In Homing While Going New Width',sRcyText:='Forward Limit Switch Is Activated. Reset The Error By Operate The Motor Backwards.'),(sAlmText:='Reverse Limit Activated In Homing While Going New Width',sRcyText:='Reverse Limit Switch Is Activated. Reset The Error By Operate The Motor Backwards.'),(sAlmText:='Forward Limit Activated In Move Absolute While Going New Width',sRcyText:='Forward Limit Switch Is Activated. Reset The Error By Operate The Motor Backwards.'),(sAlmText:='Reverse Limit Activated In Move Absolute While Going New Width',sRcyText:='Reverse Limit Switch Is Activated. Reset The Error By Operate The Motor Backwards.'),(sAlmText:='Power On Time Out While Full Homing',sRcyText:='Timeout Expired Before Operation Completed. Reset And Resume Operation.'),(sAlmText:='Homing Time Out While Full Homing',sRcyText:='Timeout Expired Before Operation Completed. Reset And Resume Operation.'),(sAlmText:='Stop Motion Time Out While Full Homing',sRcyText:='Timeout Expired Before Operation Completed. Reset And Resume Operation.'),(sAlmText:='Axis Error Reset Failed While Full Homing',sRcyText:='Axis Error Reset Failed. Please Retry Again Reset Operation. If The Problem Persists, Please Contact Nutek For A Possible Solution.'),(sAlmText:='Axis Error Occur In Homing While Full Homing',sRcyText:='Servo Motor Abnormal Operation. Reset And Resume Operation. If The Problem Persists, Please Contact Nutek For A Possible Solution.'),(sAlmText:='Homing Done But Home Flag Is Not Activated While Full Homing',sRcyText:='Servo Motor Abnormal Operation. Reset And Resume Operation. If The Problem Persists, Please Contact Nutek For A Possible Solution.'),(sAlmText:='Forward Limit Activated In Homing While Full Homing',sRcyText:='Forward Limit Switch Is Activated. Reset The Error By Operate The Motor Backwards.'),(sAlmText:='Reverse Limit Activated In Homing While Full Homing',sRcyText:='Reverse Limit Switch Is Activated. Reset The Error By Operate The Motor Backwards.'),(sAlmText:='Power On Time Out',sRcyText:='Timeout Expired Before Operation Completed. Reset And Resume Operation.'),(sAlmText:='Power Off Time Out',sRcyText:='Timeout Expired Before Operation Completed. Reset And Resume Operation.'),(sAlmText:='Homing Time Out',sRcyText:='Timeout Expired Before Operation Completed. Reset And Resume Operation.'),(sAlmText:='Move Absolute Time Out',sRcyText:='Timeout Expired Before Operation Completed. Reset And Resume Operation.'),(sAlmText:='Move Relative Time Out',sRcyText:='Timeout Expired Before Operation Completed. Reset And Resume Operation.'),(sAlmText:='Stop Motion Time Out',sRcyText:='Timeout Expired Before Operation Completed. Reset And Resume Operation.'),(sAlmText:='SDO Write Error',sRcyText:='Fail While Write Data. Reset The Error And Resume Operation.'),(sAlmText:='Request Absolute Position Out Of Range',sRcyText:='Request Absolute Position Does Not Fall Within The Expected Range.'),(sAlmText:='Inlet Sensor Interrupt Auto Width Movement',sRcyText:='Operation Stop Due To The Interruption Of Sensor While Auto Width Moving. Solve The Interruption To Resume Operation.'),(sAlmText:='Outlet Sensor Interrupt Auto Width Movement',sRcyText:='Operation Stop Due To The Interruption Of Sensor While Auto Width Moving. Solve The Interruption To Resume Operation.'),(sAlmText:='Clear Sensor Interrupt Auto Width Movement',sRcyText:='Operation Stop Due To The Interruption Of Sensor While Auto Width Moving. Solve The Interruption To Resume Operation.'),(sAlmText:='Middle Sensor Interrupt Auto Width Movement',sRcyText:='Operation Stop Due To The Interruption Of Sensor While Auto Width Moving. Solve The Interruption To Resume Operation.'),(sAlmText:='Sensor Interrupt Auto Width Movement',sRcyText:='Operation Stop Due To The Interruption Of Sensor While Auto Width Moving. Solve The Interruption To Resume Operation.'),(sAlmText:='Power On Time Out While Going New Width And Off',sRcyText:='Timeout Expired Before Operation Completed. Reset And Resume Operation.'),(sAlmText:='Homing Time Out While Going New Width And Off',sRcyText:='Timeout Expired Before Operation Completed. Reset And Resume Operation.'),(sAlmText:='Move Absolute Time Out While Going New Width And Off',sRcyText:='Timeout Expired Before Operation Completed. Reset And Resume Operation.'),(sAlmText:='Stop Motion Time Out While Going New Width And Off',sRcyText:='Timeout Expired Before Operation Completed. Reset And Resume Operation.'),(sAlmText:='Axis Error Reset Failed While Going New Width And Off',sRcyText:='Axis Error Reset Failed. Please Retry Again Reset Operation. If The Problem Persists, Please Contact Nutek For A Possible Solution.'),(sAlmText:='Axis Error Occur In Move Absolute While Going New Width And Off',sRcyText:='Servo Motor Abnormal Operation. Reset And Resume Operation. If The Problem Persists, Please Contact Nutek For A Possible Solution.'),(sAlmText:='Axis Error Occur In Homing While Going New Width And Off',sRcyText:='Servo Motor Abnormal Operation. Reset And Resume Operation. If The Problem Persists, Please Contact Nutek For A Possible Solution.'),(sAlmText:='Homing Done But Home Flag Is Not Activated While Going New Width And Off',sRcyText:='Servo Motor Abnormal Operation. Reset And Resume Operation. If The Problem Persists, Please Contact Nutek For A Possible Solution.'),(sAlmText:='Forward Limit Activated In Homing While Going New Width And Off',sRcyText:='Forward Limit Switch Is Activated. Reset The Error By Operate The Motor Backwards.'),(sAlmText:='Reverse Limit Activated In Homing While Going New Width And Off',sRcyText:='Reverse Limit Switch Is Activated. Reset The Error By Operate The Motor Backwards.'),(sAlmText:='Forward Limit Activated In Move Absolute While Going New Width And Off',sRcyText:='Forward Limit Switch Is Activated. Reset The Error By Operate The Motor Backwards.'),(sAlmText:='Reverse Limit Activated In Move Absolute While Going New Width And Off',sRcyText:='Reverse Limit Switch Is Activated. Reset The Error By Operate The Motor Backwards.'),2((sAlmText:='Sensor Interrupt Auto Width Movement',sRcyText:='Operation Stop Due To The Interruption Of Sensor While Auto Width Moving. Solve The Interruption To Resume Operation.')),249(0),(sAlmText:='Forward Limit Activated',sRcyText:='Forward Limit Switch Is Activated. Reset The Error By Operate The Motor Backwards.'),(sAlmText:='Reverse Limit Activated',sRcyText:='Reverse Limit Switch Is Activated. Reset The Error By Operate The Motor Backwards.')];
END_VAR
(**)
(*Local Output*)
VAR
	tyParamOut : tyMotionCANParamOut;
	sAxisErrTxt : STRING[80];
	bWidthPosDiff : BOOL;
	bJogOpen : BOOL;
	bJogClose : BOOL;
	bJogging : BOOL;
	bOpenSen : BOOL;
	bCloseSen : BOOL;
END_VAR
(**)
(*Local Input*)
VAR
	udiRstErr : UDINT := 0;
	bPrep : BOOL := TRUE;
	bEn : BOOL := TRUE;
	bDis : BOOL := FALSE;
	bOps : BOOL := FALSE;
	bManual : BOOL := FALSE;
	diWidthAtHmPos : DINT := 400;
	tyTuning : tyMotionCANTuning;
	diGoWidth : DINT := 150;
	diJogVelInUMPS : DINT := 10000;
	diMovePosInUM : DINT := 0;
	diMoveDistInUM : DINT := 0;
	diMoveVelInUMPS : DINT := 10000;
	diMoveAcc : DINT := 500;
	diMoveDec : DINT := 500;
	diMinAbsPosInUM : DINT := -3000;
	diMaxAbsPosInUM : DINT := 10000000;
	diMinWidthInUM : DINT := 70000;
	diMaxWidthInUM : DINT := 460000;
	diWidthOffsetInUM : DINT := 0;
	bInletSensor : BOOL;
	bOutletSensor : BOOL;
	bClearSensor : BOOL;
	bMiddleSensor : BOOL;
	bInterruptSensor : BOOL;
	bOpenInterruptSensor : BOOL;
	bCloseInterruptSensor : BOOL;
	bDir : BOOL;
	bDirBl : BOOL;
	bNoIndexPulse : BOOL;
	usiNode : USINT;
	sDevice : STRING[3];
	sProgNm : STRING[15] := 'AWOpen';
	diMoveBacklashDistInUM : DINT := 3000;
	diPitchInUM : DINT := 3000;
	tyParamInHm : tyMotionCANParamInHm;
	tyParamInConvert : tyMotionCANParamInConvert := (diPitchInUM:=3000);
	bNtSettingsLoadDone : BOOL := TRUE;
	eMotorType : eServoMotorType := DeltaAsdaA2;
END_VAR
(**)
(*Local*)
VAR
	bRstErr : BOOL;
	udiRstErrOld : UDINT;
	bInitDone : BOOL;
	bInitialDone : BOOL;
	bModuleOKChk : BOOL := TRUE;
	bModuleOK : BOOL;
	bModuleNotOK : BOOL := TRUE;
	bModuleNotOKLock : BOOL;
	bNotInterruptible : BOOL;
	bInterruptSensor1 : BOOL;
	bInterruptSensor2 : BOOL;
	diActualPosInUMOld : DINT;
	usiRstStep : USINT := 0;
	usiStep : USINT;
	usiCount : USINT;
	fbTm : TON := (PT:=T#2s);
	fbServoModuleNotOk : TON := (IN:=FALSE,PT:=T#2s);
	fbServoModuleOk : TON := (IN:=FALSE,PT:=T#5s);
	fbRstNodeTimer : TON := (PT:=T#3s);
	tyParamInMove : tyMotionCANParamInMove;
	tyParamInDriver : tyMotionCANDriverIn;
	tyParamOutDriver : tyMotionCANDriverOut := (siModOfOpt_6060:=6);
	fbStop : fbMotionCANStop;
	fbRstAxisErr : fbMotionCANRstAxisErr;
	fbJog : fbMotionCANJog;
	fbMovRel : fbMotionCANMovRel;
	fbMovAbs : fbMotionCANMovAbs;
	fbHoming : fbMotionCANHoming;
	fbPwrOff : fbMotionCANPwrOff;
	fbPwrOn : fbMotionCANPwrOn;
	fbFullHm : fbMotionCANFullHm;
	fbFullMovAbs : fbMotionCANFullMovAbs;
	fbFullMovAbsBl : fbMotionCANFullMovAbsBl;
	fbModuleOK : fbMotionCANModuleOK;
	fbSDOWrite : fbCANSDOWriteArrayParam;
	udiModuleNum : UDINT := 1;
END_VAR
```

### AWPushOrPuller.var - Change By Project
```iecst
(*2019-04-24*)
(**)
(*Action & State & Status*)
VAR
	p_AWPushOrPullerStat : UDINT;
	p_AWPushOrPullerStatus : UDINT;
	p_AWPushOrPullerStatTxt : UDINT;
END_VAR
(**)
(*Alarm*)
VAR
	p_AWPushOrPullerAlmData : UDINT;
	p_AWPushOrPullerAlmData1 : UDINT;
	p_AWPushOrPullerAlmData2 : UDINT;
	p_AWPushOrPullerAlmData3 : UDINT;
END_VAR
(**)
(*Output*)
VAR
	p_AWPushOrPullerParamOut : UDINT;
	p_AWPushOrPullerPwrOn : UDINT;
	p_AWPushOrPullerIsHomed : UDINT;
	p_AWPushOrPullerPosDiff : UDINT;
	p_AWPushOrPullerAxisErr : UDINT;
	p_AWPushOrPullerAxisErrID : UDINT;
	p_AWPushOrPullerAxisErrTxt : UDINT;
	p_AWPushOrPullerFwdLmtSen : UDINT;
	p_AWPushOrPullerRevLmtSen : UDINT;
	p_AWPushOrPullerActualPos : UDINT;
	p_AWPushOrPullerWidthPosDiff : UDINT;
	p_AWPushOrPullerJogging : UDINT;
	p_AWPushOrPullerOpenSen : UDINT;
	p_AWPushOrPullerCloseSen : UDINT;
END_VAR
```

### Program Logical/CANOpenServo/AW/AWPushOrPuller (IEC, version 1.00.0) - 1.00.0 - NtMotion v5.00.0

#### Init.st - Change By Project
```iecst
(** 2019-04-24 **)
PROGRAM _INIT

	(* Always Change If Project Change *)

	//Pass Address To Global Address For External Use
	//Action, State & Status
	p_AWPushOrPullerStat		:= ADR(eStat);
	p_AWPushOrPullerStatus		:= ADR(eMainStatus);
	p_AWPushOrPullerStatTxt		:= ADR(sStatTxt);

	//Alarm
	p_AWPushOrPullerAlmData		:= ADR(tyAlmData);
	p_AWPushOrPullerAlmData1	:= ADR(tyAlmData1);
	p_AWPushOrPullerAlmData2	:= ADR(tyAlmData2);
	p_AWPushOrPullerAlmData3	:= ADR(tyAlmData3);

	//Output
	p_AWPushOrPullerParamOut		:= ADR(tyParamOut);
	p_AWPushOrPullerPwrOn			:= ADR(tyParamOut.bPwrOn);
	p_AWPushOrPullerIsHomed			:= ADR(tyParamOut.bIsHomed);
	p_AWPushOrPullerPosDiff			:= ADR(tyParamOut.bPosDiff);
	p_AWPushOrPullerAxisErr			:= ADR(tyParamOut.bAxisErr);
	p_AWPushOrPullerAxisErrID		:= ADR(tyParamOut.udiAxisErrID);
	p_AWPushOrPullerFwdLmtSen		:= ADR(tyParamOut.bFwdLmtSen);
	p_AWPushOrPullerRevLmtSen		:= ADR(tyParamOut.bRevLmtSen);
	p_AWPushOrPullerActualPos		:= ADR(tyParamOut.diActualPosInUM);
	p_AWPushOrPullerAxisErrTxt		:= ADR(sAxisErrTxt);
	p_AWPushOrPullerWidthPosDiff	:= ADR(bWidthPosDiff);
	p_AWPushOrPullerJogging			:= ADR(bJogging);
	p_AWPushOrPullerOpenSen			:= ADR(bOpenSen);
	p_AWPushOrPullerCloseSen		:= ADR(bCloseSen);

	(* Always Change If Project Change *)

END_PROGRAM
```

#### Act_InitGlobal.st - Change By Project
```iecst
(** 2019-04-09 **)
ACTION Act_InitGlobal:

	(* Always Change If Project Change *)

	//Pass Data To Link
	p_bLinkOpsRun ACCESS p_OpsRun;
	p_bLinkStartupRun ACCESS p_StartupRun;
	p_diLinkProdSelWidth ACCESS p_ProdRcpCurrRcp1Width;
	p_diLinkPshrOffset ACCESS p_ProdRcpCurrRcp1PshrPulerOffset;
	p_diLinkMnlGoWidth ACCESS p_UIMnlAWPushOrPullerGoWidth;
	p_bLinkSafetyRelay ACCESS p_DISafetyRlySig;

	//Pass Data To Internal Use
	p_udiRstErr ACCESS p_RstErrReset;
	p_bManual ACCESS p_UIMnlMod;
	p_bPrep ACCESS p_NtParamAWPushPulPrep;
	p_bDis ACCESS p_McParamAWPusherDis;
	p_bOps ACCESS p_OpsStatusRun;
	p_diWidthAtHmPos ACCESS p_McParamAWPusherAtHmPos;
	p_tyTuning ACCESS p_NtParamAWPushPulTuning;
	p_diJogVelInUMPS ACCESS p_UIMnlAWPushOrPullerJogSpd;
	p_diMovePosInUM ACCESS p_UIMnlAWPushOrPullerTargetPos;
	p_diMoveDistInUM ACCESS p_UIMnlAWPushOrPullerStepSize;
	p_diMoveAcc ACCESS p_NtParamAWPushPulAcc;
	p_diMoveDec ACCESS p_NtParamAWPushPulDec;
	p_diMinWidthInUM ACCESS p_NtParamProdRcpMinWidth;
	p_diMaxWidthInUM ACCESS p_NtParamProdRcpMaxWidth;
	p_diWidthOffsetInUM ACCESS p_NtParamPushPulAWidthOffset;
	p_bInletSensor ACCESS p_DIConvLftSen;
	p_bOutletSensor ACCESS p_DIConvRgtSen;
	p_bDir ACCESS p_NtParamAWPushPulDir;
	p_bDirBl ACCESS p_NtParamAWPushPulDirBl;
	p_usiNode ACCESS p_NtParamAWPushPulNode;
	p_sDevice ACCESS p_NtParamAWPushPulDevice;
	p_sProgNm ACCESS p_NtParamAWPushPulProgNm;
	p_diMoveBacklashDistInUM ACCESS p_NtParamAWPushPulMovBlDistInUM;
	p_diPitchInUM ACCESS p_NtParamAWPushPulPitchInUM;
	p_tyParamInHm ACCESS p_NtParamAWPushPulParamInHm;
	p_tyParamInConvert ACCESS p_NtParamAWPushPulParamInConvert;
	p_bNtSettingsLoadDone ACCESS p_StartupNtSettingsLoadDone;
	p_eNtParamMotorType ACCESS p_NtParamAWPushPulMotorType;

	p_bInletShutterCloseRS ACCESS p_DIInShutterCloseRS;
	p_bOutletShutterCloseRS ACCESS p_DIOutShutterCloseRS;
	p_bOutletShutterCloseRS2 ACCESS p_DIOutShutterCloseRS2;
	p_bOutletShutterCloseRS3 ACCESS p_DIOutShutterCloseRS3;
	p_bProjInletShutPrep ACCESS p_NtParamProjInletShutPrep;
	p_bInShutterDis ACCESS p_McParamInShutterDis;
	p_bProjOutletShutPrep ACCESS p_NtParamProjOutletShutPrep;

	p_bPusherRetSen ACCESS p_DIPusherRetRS;
	p_bPusherExtSen ACCESS p_DIPusherExtRS;
	(* Always Change If Project Change *)

END_ACTION
```

#### InputRef_Link.var - Change By Project
```iecst
(*2019-04-09*)
(**)
VAR
	p_bLinkOpsRun : REFERENCE TO BOOL;
	p_bLinkStartupRun : REFERENCE TO BOOL;
	p_diLinkProdSelWidth : REFERENCE TO DINT;
	p_diLinkPshrOffset : REFERENCE TO DINT;
	p_diLinkMnlGoWidth : REFERENCE TO DINT;
	p_bLinkSafetyRelay : REFERENCE TO BOOL;
END_VAR
```

#### Act_LinkAction.st - Change By Project
```iecst
(** 2019-10-21 **)
ACTION Act_LinkAction:

	IF eStatus = Idle THEN
		IF bModuleNotOK THEN
			p_eAct ACCESS ADR(eAct);
		ELSE
			IF p_bLinkStartupRun = TRUE THEN
				p_eAct ACCESS p_StartupAWPushPulAct;
			ELSIF p_bLinkOpsRun = TRUE THEN
				p_eAct ACCESS p_OpsTravLifULAWPushPullAct;
			ELSIF p_bManual = TRUE THEN
				p_eAct ACCESS p_UIAWPushOrPullerAct;
			ELSE
				p_eAct ACCESS ADR(eAct);
			END_IF
		END_IF
	END_IF

	IF EDGENEG(p_bManual) OR EDGENEG(p_bLinkOpsRun) OR EDGENEG(p_bLinkStartupRun) THEN
		tyParamOutDriver.uiCtrlword_6040	:= 0;
	END_IF

END_ACTION
```

#### Act_Link.st - Change By Project
```iecst
(** 2019-03-29 **)
ACTION Act_Link:

	IF p_bManual = TRUE THEN
		p_diMoveVelInUMPS ACCESS p_UIMnlAWPushOrPullerNomSpd;
		IF p_diLinkMnlGoWidth < p_diWidthAtHmPos THEN
			p_diGoWidth := p_diWidthAtHmPos;
		ELSE
			p_diGoWidth	:= p_diLinkMnlGoWidth;
		END_IF

	ELSE
		p_diGoWidth := (p_diLinkProdSelWidth/2) + p_diLinkPshrOffset;

		p_diMoveVelInUMPS ACCESS p_NtParamAWPushPulAutoSpd;

		IF p_diGoWidth <= p_diWidthAtHmPos THEN
			p_diGoWidth := p_diWidthAtHmPos + 3000;
		ELSE
			p_diGoWidth := (p_diLinkProdSelWidth/2) + p_diLinkPshrOffset;

		END_IF

	END_IF

	IF p_bProjInletShutPrep = TRUE AND p_bInShutterDis = FALSE AND (p_bOps OR p_bManual) THEN
		IF (p_bInletShutterCloseRS = FALSE AND NOT p_bOps) OR p_bPusherRetSen = FALSE OR p_bPusherExtSen THEN
			bInterruptSensor1 := TRUE;
		ELSE
			bInterruptSensor1 := FALSE;
		END_IF
	ELSE
		bInterruptSensor1 := FALSE;
	END_IF

	IF p_bProjOutletShutPrep = TRUE AND (p_bOps OR p_bManual)THEN
		IF ((p_bOutletShutterCloseRS = FALSE OR p_bOutletShutterCloseRS2 = FALSE OR p_bOutletShutterCloseRS3 = FALSE) AND NOT p_bOps) OR p_bPusherRetSen = FALSE OR p_bPusherExtSen THEN
			bInterruptSensor2 := TRUE;
		ELSE
			bInterruptSensor2 := FALSE;
		END_IF
	ELSE
		bInterruptSensor2 := FALSE;
	END_IF

	IF NOT p_bOps THEN
		bInterruptSensor1	:= FALSE;
		bInterruptSensor2   := FALSE;
		p_bInterruptSensor	:= FALSE;
	END_IF

	p_bInterruptSensor := bInterruptSensor2 OR bInterruptSensor1;

END_ACTION
```

#### Act_Initial.st - Do Not Change!!!
```iecst
(** 2020-03-16 **)
ACTION Act_Initial:

	//Initial
	sStatTxt	:= a_sStatText[eStat];

	tyParamInMove.diBacklashDistInUM	:= p_diMoveBacklashDistInUM;
	tyParamInMove.diAcc					:= p_diMoveAcc;
	tyParamInMove.diDec					:= p_diMoveDec;

	//p_tyParamInConvert.diPitchInUM	:= fPitchCalc(p_diWidthOffsetInUM , p_diMaxWidthInUM , p_diMinWidthInUM , p_diPitchInUM);

	fbModuleOK.sDevice	:= p_sDevice;
	fbModuleOK.usiNode	:= p_usiNode;
	fbModuleOK.tDlyTm	:= T#5s;
	fbModuleOK(bEn := FALSE);

	fbSDOWrite.sDevice	:= p_sDevice;
	fbSDOWrite.usiNode	:= p_usiNode;
	fbSDOWrite.eMotorType	:= p_eNtParamMotorType;
	fbSDOWrite(bEn := FALSE);

	fbFullMovAbsBl.p_tyParamOutDriver				:= ADR(tyParamOutDriver);
	fbFullMovAbsBl.tyParamInMove.diBacklashDistInUM	:= p_diMoveBacklashDistInUM;
	fbFullMovAbsBl.tyParamInMove.diAcc				:= p_diMoveAcc;
	fbFullMovAbsBl.tyParamInMove.diDec				:= p_diMoveDec;
	//fbFullMovAbsBl.tyParamInConvert					:= p_tyParamInConvert;
	fbFullMovAbsBl.bDir								:= p_bDir;
	fbFullMovAbsBl.bDirBl							:= p_bDirBl;
	fbFullMovAbsBl.bNoIndexPulse					:= p_bNoIndexPulse;
	fbFullMovAbsBl.eMotorType						:= p_eNtParamMotorType;
	fbFullMovAbsBl(bEn := FALSE);

	fbFullMovAbs.p_tyParamOutDriver					:= ADR(tyParamOutDriver);
	fbFullMovAbs.bDir								:= p_bDir;
	fbFullMovAbs.bNoIndexPulse						:= p_bNoIndexPulse;
	fbFullMovAbs.eMotorType							:= p_eNtParamMotorType;
	fbFullMovAbs(bEn := FALSE);

	fbFullHm.p_tyParamOutDriver	:= ADR(tyParamOutDriver);
	fbFullHm.bDir				:= p_bDir;
	fbFullHm.bNoIndexPulse		:= p_bNoIndexPulse;
	fbFullHm.eMotorType			:= p_eNtParamMotorType;
	fbFullHm(bEn := FALSE);

	fbPwrOn.p_tyParamOutDriver	:= ADR(tyParamOutDriver);
	fbPwrOn.eMotorType			:= p_eNtParamMotorType;
	fbPwrOn(bEn := FALSE);

	fbPwrOff.p_tyParamOutDriver	:= ADR(tyParamOutDriver);
	fbPwrOff.eMotorType			:= p_eNtParamMotorType;
	fbPwrOff(bEn := FALSE);

	fbHoming.p_tyParamOutDriver	:= ADR(tyParamOutDriver);
	fbHoming.bDir				:= p_bDir;
	fbHoming.bNoIndexPulse		:= p_bNoIndexPulse;
	fbHoming.eMotorType			:= p_eNtParamMotorType;
	fbHoming(bEn := FALSE);

	fbMovAbs.p_tyParamOutDriver					:= ADR(tyParamOutDriver);
	fbMovAbs.tyParamInMove.diBacklashDistInUM	:= p_diMoveBacklashDistInUM;
	fbMovAbs.tyParamInMove.diAcc				:= p_diMoveAcc;
	fbMovAbs.tyParamInMove.diDec				:= p_diMoveDec;
	fbMovAbs.tyParamInConvert					:= p_tyParamInConvert;
	fbMovAbs.bDir								:= p_bDir;
	fbMovAbs.eMotorType							:= p_eNtParamMotorType;
	fbMovAbs(bEn := FALSE);

	fbMovRel.p_tyParamOutDriver					:= ADR(tyParamOutDriver);
	fbMovRel.tyParamInMove.diBacklashDistInUM	:= p_diMoveBacklashDistInUM;
	fbMovRel.tyParamInMove.diAcc				:= p_diMoveAcc;
	fbMovRel.tyParamInMove.diDec				:= p_diMoveDec;
	fbMovRel.tyParamInConvert					:= p_tyParamInConvert;
	fbMovRel.bDir								:= p_bDir;
	fbMovRel.eMotorType							:= p_eNtParamMotorType;
	fbMovRel(bEn := FALSE);

	fbJog.p_tyParamOutDriver	:= ADR(tyParamOutDriver);
	fbJog.tyParamInConvert		:= p_tyParamInConvert;
	fbJog.eMotorType			:= p_eNtParamMotorType;
	fbJog(bEn := FALSE);

	fbRstAxisErr.p_tyParamOutDriver	:= ADR(tyParamOutDriver);
	fbRstAxisErr(bEn := FALSE);

	fbStop.p_tyParamOutDriver	:= ADR(tyParamOutDriver);
	fbStop(bEn := FALSE);

	bModuleNotOK	:= TRUE;

END_ACTION
```
